LIN {X 0,Y 564.542,Z 419.185,A -85,B 0,C 180,E1 24922.898,E2 24922.898} C_VEL
LIN {X 0,Y 566.553,Z 422.727,A -85,B 0,C 180,E1 24922.507,E2 24922.507} C_VEL
LIN {X 0,Y 580.883,Z 441.824,A -85,B 0,C 180,E1 24920.03,E2 24920.03} C_VEL
LIN {X 0,Y 586.064,Z 449.548,A -85,B 0,C 180,E1 24919.171,E2 24919.171} C_VEL
LIN {X 0,Y 576.668,Z 659.273,A -85,B 0,C 180,E1 24915.972,E2 24915.972} C_VEL
LIN {X 0,Y 572.189,Z 766.018,A -85,B 0,C 180,E1 24914.357,E2 24914.357} C_VEL
LIN {X 0,Y 570.088,Z 794.768,A -85,B 0,C 180,E1 24913.761,E2 24913.761} C_VEL
LIN {X 0,Y 567.768,Z 818.372,A -85,B 0,C 180,E1 24913.108,E2 24913.108} C_VEL
LIN {X 0,Y 565.366,Z 838.963,A -85,B 0,C 180,E1 24912.414,E2 24912.414} C_VEL
LIN {X 0,Y 562.569,Z 859.83,A -85,B 0,C 180,E1 24911.584,E2 24911.584} C_VEL
LIN {X 0,Y 558.94,Z 883.872,A -85,B 0,C 180,E1 24910.457,E2 24910.457} C_VEL
LIN {X 0,Y 554.622,Z 908.25,A -85,B 0,C 180,E1 24909.087,E2 24909.087} C_VEL
LIN {X 0,Y 551.08,Z 926.843,A -85,B 0,C 180,E1 24907.884,E2 24907.884} C_VEL
LIN {X 0,Y 547.473,Z 944.537,A -85,B 0,C 180,E1 24906.595,E2 24906.595} C_VEL
LIN {X 0,Y 543.684,Z 962.173,A -85,B 0,C 180,E1 24905.151,E2 24905.151} C_VEL
LIN {X 0,Y 538.855,Z 983.671,A -85,B 0,C 180,E1 24903.145,E2 24903.145} C_VEL
LIN {X 0,Y 534.335,Z 1002.75,A -85,B 0,C 180,E1 24901.078,E2 24901.078} C_VEL
LIN {X 0,Y 530.36,Z 1019.387,A -85,B 0,C 180,E1 24899.024,E2 24899.024} C_VEL
LIN {X 0,Y 526.19,Z 1036.957,A -85,B 0,C 180,E1 24896.534,E2 24896.534} C_VEL
LIN {X 0,Y 522.376,Z 1053.129,A -85,B 0,C 180,E1 24893.876,E2 24893.876} C_VEL
LIN {X 0,Y 519.153,Z 1069.381,A -85,B 0,C 180,E1 24890.912,E2 24890.912} C_VEL
LIN {X 0,Y 516.803,Z 1082.675,A -85,B 0,C 180,E1 24888.127,E2 24888.127} C_VEL
LIN {X 0,Y 514.982,Z 1094.284,A -85,B 0,C 180,E1 24885.286,E2 24885.286} C_VEL
LIN {X 0,Y 513.617,Z 1104.724,A -85,B 0,C 180,E1 24882.289,E2 24882.289} C_VEL
LIN {X 0,Y 512.807,Z 1113.008,A -85,B 0,C 180,E1 24879.455,E2 24879.455} C_VEL
LIN {X 0,Y 512.269,Z 1120.002,A -85,B 0,C 180,E1 24876.47,E2 24876.47} C_VEL
LIN {X 0,Y 512.013,Z 1125.314,A -85,B 0,C 180,E1 24873.55,E2 24873.55} C_VEL
LIN {X 0,Y 511.941,Z 1128.909,A -85,B 0,C 180,E1 24870.779,E2 24870.779} C_VEL
LIN {X 0,Y 511.913,Z 1131.135,A -85,B 0,C 180,E1 24867.955,E2 24867.955} C_VEL
LIN {X 0,Y 511.904,Z 1131.984,A -85,B 0,C 180,E1 24865.079,E2 24865.079} C_VEL
LIN {X 0,Y 511.904,Z 1131.233,A -85,B 0,C 180,E1 24862.147,E2 24862.147} C_VEL
LIN {X 0,Y 511.939,Z 1129.064,A -85,B 0,C 180,E1 24859.274,E2 24859.274} C_VEL
LIN {X 0,Y 512.001,Z 1125.626,A -85,B 0,C 180,E1 24856.566,E2 24856.566} C_VEL
LIN {X 0,Y 512.205,Z 1120.709,A -85,B 0,C 180,E1 24853.778,E2 24853.778} C_VEL
LIN {X 0,Y 512.707,Z 1114.184,A -85,B 0,C 180,E1 24850.904,E2 24850.904} C_VEL
LIN {X 0,Y 513.531,Z 1105.747,A -85,B 0,C 180,E1 24847.946,E2 24847.946} C_VEL
LIN {X 0,Y 514.839,Z 1095.333,A -85,B 0,C 180,E1 24844.902,E2 24844.902} C_VEL
LIN {X 0,Y 516.649,Z 1083.593,A -85,B 0,C 180,E1 24841.996,E2 24841.996} C_VEL
LIN {X 0,Y 518.987,Z 1070.357,A -85,B 0,C 180,E1 24839.185,E2 24839.185} C_VEL
LIN {X 0,Y 523.302,Z 1049.733,A -85,B 0,C 180,E1 24835.397,E2 24835.397} C_VEL
LIN {X 0,Y 527.1,Z 1034.636,A -85,B 0,C 180,E1 24832.917,E2 24832.917} C_VEL
LIN {X 0,Y 530.836,Z 1019.658,A -85,B 0,C 180,E1 24830.787,E2 24830.787} C_VEL
LIN {X 0,Y 534.371,Z 1005.434,A -85,B 0,C 180,E1 24828.997,E2 24828.997} C_VEL
LIN {X 0,Y 537.967,Z 990.583,A -85,B 0,C 180,E1 24827.331,E2 24827.331} C_VEL
LIN {X 0,Y 542.61,Z 970.761,A -85,B 0,C 180,E1 24825.377,E2 24825.377} C_VEL
LIN {X 0,Y 546.709,Z 951.555,A -85,B 0,C 180,E1 24823.75,E2 24823.75} C_VEL
LIN {X 0,Y 550.21,Z 934.054,A -85,B 0,C 180,E1 24822.442,E2 24822.442} C_VEL
LIN {X 0,Y 553.849,Z 914.316,A -85,B 0,C 180,E1 24821.146,E2 24821.146} C_VEL
LIN {X 0,Y 557.856,Z 889.499,A -85,B 0,C 180,E1 24819.761,E2 24819.761} C_VEL
LIN {X 0,Y 560.615,Z 869.773,A -85,B 0,C 180,E1 24818.828,E2 24818.828} C_VEL
LIN {X 0,Y 562.93,Z 850.518,A -85,B 0,C 180,E1 24818.044,E2 24818.044} C_VEL
LIN {X 0,Y 565.079,Z 829.301,A -85,B 0,C 180,E1 24817.31,E2 24817.31} C_VEL
LIN {X 0,Y 567.288,Z 800.913,A -85,B 0,C 180,E1 24816.536,E2 24816.536} C_VEL
LIN {X 0,Y 568.472,Z 778.885,A -85,B 0,C 180,E1 24816.082,E2 24816.082} C_VEL
LIN {X 0,Y 574.153,Z 658.763,A -85,B 0,C 180,E1 24814.166,E2 24814.166} C_VEL
LIN {X 0,Y 579.443,Z 579.746,A -85,B 0,C 180,E1 24812.805,E2 24812.805} C_VEL
LIN {X 0,Y 586.189,Z 505.599,A -85,B 0,C 180,E1 24811.443,E2 24811.443} C_VEL
LIN {X 0,Y 592.771,Z 449.982,A -85,B 0,C 180,E1 24810.35,E2 24810.35} C_VEL
LIN {X 0,Y 591.734,Z 444.986,A -85,B 0,C 180,E1 24809.456,E2 24809.456} C_VEL
LIN {X 0,Y 591.658,Z 444.729,A -85,B 0,C 180,E1 24809.362,E2 24809.362} C_VEL
LIN {X 0,Y 589.852,Z 450.751,A -85,B 0,C 180,E1 24808.449,E2 24808.449} C_VEL
LIN {X 0,Y 588.941,Z 461.125,A -85,B 0,C 180,E1 24807.237,E2 24807.237} C_VEL
LIN {X 0,Y 589.012,Z 464.19,A -85,B 0,C 180,E1 24806.908,E2 24806.908} C_VEL
LIN {X 0,Y 588.095,Z 484.724,A -85,B 0,C 180,E1 24805.902,E2 24805.902} C_VEL
LIN {X 0,Y 588.06,Z 490.969,A -85,B 0,C 180,E1 24805.601,E2 24805.601} C_VEL
LIN {X 0,Y 581.292,Z 561.279,A -85,B 0,C 180,E1 24804.259,E2 24804.259} C_VEL
LIN {X 0,Y 575.759,Z 638.702,A -85,B 0,C 180,E1 24802.87,E2 24802.87} C_VEL
LIN {X 0,Y 570.578,Z 738.854,A -85,B 0,C 180,E1 24801.211,E2 24801.211} C_VEL
LIN {X 0,Y 565.248,Z 887.623,A -85,B 0,C 180,E1 24798.952,E2 24798.952} C_VEL
LIN {X 0,Y 563.149,Z 916.285,A -85,B 0,C 180,E1 24798.378,E2 24798.378} C_VEL
LIN {X 0,Y 560.931,Z 940.423,A -85,B 0,C 180,E1 24797.778,E2 24797.778} C_VEL
LIN {X 0,Y 558.001,Z 968.794,A -85,B 0,C 180,E1 24796.91,E2 24796.91} C_VEL
LIN {X 0,Y 554.811,Z 996.1,A -85,B 0,C 180,E1 24795.867,E2 24795.867} C_VEL
LIN {X 0,Y 552.139,Z 1017.393,A -85,B 0,C 180,E1 24794.921,E2 24794.921} C_VEL
LIN {X 0,Y 549.242,Z 1038.814,A -85,B 0,C 180,E1 24793.843,E2 24793.843} C_VEL
LIN {X 0,Y 546.178,Z 1060.331,A -85,B 0,C 180,E1 24792.613,E2 24792.613} C_VEL
LIN {X 0,Y 542.506,Z 1085.129,A -85,B 0,C 180,E1 24791.005,E2 24791.005} C_VEL
LIN {X 0,Y 538.667,Z 1108.867,A -85,B 0,C 180,E1 24789.22,E2 24789.22} C_VEL
LIN {X 0,Y 535.764,Z 1126.329,A -85,B 0,C 180,E1 24787.744,E2 24787.744} C_VEL
LIN {X 0,Y 533.088,Z 1142.045,A -85,B 0,C 180,E1 24786.282,E2 24786.282} C_VEL
LIN {X 0,Y 530.41,Z 1157.572,A -85,B 0,C 180,E1 24784.701,E2 24784.701} C_VEL
LIN {X 0,Y 527.7,Z 1173.227,A -85,B 0,C 180,E1 24782.943,E2 24782.943} C_VEL
LIN {X 0,Y 525.229,Z 1187.423,A -85,B 0,C 180,E1 24781.185,E2 24781.185} C_VEL
LIN {X 0,Y 523.309,Z 1198.436,A -85,B 0,C 180,E1 24779.661,E2 24779.661} C_VEL
LIN {X 0,Y 520.705,Z 1211.245,A -85,B 0,C 180,E1 24777.481,E2 24777.481} C_VEL
LIN {X 0,Y 518.448,Z 1222.98,A -85,B 0,C 180,E1 24775.228,E2 24775.228} C_VEL
LIN {X 0,Y 516.666,Z 1233.28,A -85,B 0,C 180,E1 24773.012,E2 24773.012} C_VEL
LIN {X 0,Y 515.063,Z 1243.808,A -85,B 0,C 180,E1 24770.452,E2 24770.452} C_VEL
LIN {X 0,Y 513.624,Z 1254.739,A -85,B 0,C 180,E1 24767.328,E2 24767.328} C_VEL
LIN {X 0,Y 512.851,Z 1262.137,A -85,B 0,C 180,E1 24764.797,E2 24764.797} C_VEL
LIN {X 0,Y 512.406,Z 1267.799,A -85,B 0,C 180,E1 24762.509,E2 24762.509} C_VEL
LIN {X 0,Y 512.121,Z 1272.693,A -85,B 0,C 180,E1 24760.12,E2 24760.12} C_VEL
LIN {X 0,Y 511.965,Z 1276.677,A -85,B 0,C 180,E1 24757.632,E2 24757.632} C_VEL
LIN {X 0,Y 511.924,Z 1279.659,A -85,B 0,C 180,E1 24755.038,E2 24755.038} C_VEL
LIN {X 0,Y 511.911,Z 1281.599,A -85,B 0,C 180,E1 24752.015,E2 24752.015} C_VEL
LIN {X 0,Y 511.865,Z 1281.871,A -85,B 0,C 180,E1 24749.328,E2 24749.328} C_VEL
LIN {X 0,Y 511.909,Z 1281.082,A -85,B 0,C 180,E1 24746.977,E2 24746.977} C_VEL
LIN {X 0,Y 511.93,Z 1279.199,A -85,B 0,C 180,E1 24744.508,E2 24744.508} C_VEL
LIN {X 0,Y 511.97,Z 1276.356,A -85,B 0,C 180,E1 24742.142,E2 24742.142} C_VEL
LIN {X 0,Y 512.156,Z 1272.279,A -85,B 0,C 180,E1 24739.653,E2 24739.653} C_VEL
LIN {X 0,Y 512.544,Z 1266.27,A -85,B 0,C 180,E1 24736.806,E2 24736.806} C_VEL
LIN {X 0,Y 513.279,Z 1257.914,A -85,B 0,C 180,E1 24733.709,E2 24733.709} C_VEL
LIN {X 0,Y 514.226,Z 1249.696,A -85,B 0,C 180,E1 24731.169,E2 24731.169} C_VEL
LIN {X 0,Y 515.454,Z 1241.06,A -85,B 0,C 180,E1 24728.851,E2 24728.851} C_VEL
LIN {X 0,Y 517.115,Z 1230.712,A -85,B 0,C 180,E1 24726.406,E2 24726.406} C_VEL
LIN {X 0,Y 519.818,Z 1215.891,A -85,B 0,C 180,E1 24723.373,E2 24723.373} C_VEL
LIN {X 0,Y 522.446,Z 1202.553,A -85,B 0,C 180,E1 24721.002,E2 24721.002} C_VEL
LIN {X 0,Y 524.453,Z 1192.013,A -85,B 0,C 180,E1 24719.4,E2 24719.4} C_VEL
LIN {X 0,Y 527.516,Z 1175.905,A -85,B 0,C 180,E1 24717.238,E2 24717.238} C_VEL
LIN {X 0,Y 530.602,Z 1160.006,A -85,B 0,C 180,E1 24715.313,E2 24715.313} C_VEL
LIN {X 0,Y 534.437,Z 1140.647,A -85,B 0,C 180,E1 24713.203,E2 24713.203} C_VEL
LIN {X 0,Y 538.764,Z 1118.423,A -85,B 0,C 180,E1 24711.082,E2 24711.082} C_VEL
LIN {X 0,Y 542.437,Z 1099.473,A -85,B 0,C 180,E1 24709.476,E2 24709.476} C_VEL
LIN {X 0,Y 546.072,Z 1080.345,A -85,B 0,C 180,E1 24708.023,E2 24708.023} C_VEL
LIN {X 0,Y 550.322,Z 1057.451,A -85,B 0,C 180,E1 24706.48,E2 24706.48} C_VEL
LIN {X 0,Y 554.631,Z 1032.424,A -85,B 0,C 180,E1 24705.034,E2 24705.034} C_VEL
LIN {X 0,Y 558.14,Z 1010.377,A -85,B 0,C 180,E1 24703.932,E2 24703.932} C_VEL
LIN {X 0,Y 561.113,Z 990.283,A -85,B 0,C 180,E1 24703.063,E2 24703.063} C_VEL
LIN {X 0,Y 564.037,Z 968.586,A -85,B 0,C 180,E1 24702.259,E2 24702.259} C_VEL
LIN {X 0,Y 567.292,Z 941.486,A -85,B 0,C 180,E1 24701.432,E2 24701.432} C_VEL
LIN {X 0,Y 569.778,Z 915.224,A -85,B 0,C 180,E1 24700.824,E2 24700.824} C_VEL
LIN {X 0,Y 571.357,Z 892.816,A -85,B 0,C 180,E1 24700.418,E2 24700.418} C_VEL
LIN {X 0,Y 580.407,Z 670.692,A -85,B 0,C 180,E1 24697.065,E2 24697.065} C_VEL
LIN {X 0,Y 588.793,Z 490.152,A -85,B 0,C 180,E1 24694.268,E2 24694.268} C_VEL
LIN {X 0,Y 585.464,Z 469.461,A -85,B 0,C 180,E1 24693.362,E2 24693.362} C_VEL
LIN {X 0,Y 573.553,Z 450.96,A -85,B 0,C 180,E1 24691.241,E2 24691.241} C_VEL
LIN {X 0,Y 560.617,Z 432.091,A -85,B 0,C 180,E1 24688.758,E2 24688.758} C_VEL
LIN {X 0,Y 549.882,Z 417.05,A -85,B 0,C 180,E1 24686.514,E2 24686.514} C_VEL
LIN {X 0,Y 542.341,Z 406.72,A -85,B 0,C 180,E1 24684.828,E2 24684.828} C_VEL
LIN {X 0,Y 539.641,Z 402.462,A -85,B 0,C 180,E1 24684.056,E2 24684.056} C_VEL
LIN {X 0,Y 534.084,Z 392.609,A -85,B 0,C 180,E1 24681.874,E2 24681.874} C_VEL
LIN {X 0,Y 531.056,Z 387.284,A -85,B 0,C 180,E1 24680.615,E2 24680.615} C_VEL
LIN {X 0,Y 528.6,Z 382.928,A -85,B 0,C 180,E1 24679.561,E2 24679.561} C_VEL
LIN {X 0,Y 525.714,Z 377.911,A -85,B 0,C 180,E1 24678.29,E2 24678.29} C_VEL
LIN {X 0,Y 523.432,Z 373.779,A -85,B 0,C 180,E1 24677.223,E2 24677.223} C_VEL
LIN {X 0,Y 520.587,Z 369.323,A -85,B 0,C 180,E1 24675.942,E2 24675.942} C_VEL
LIN {X 0,Y 519.744,Z 367.693,A -85,B 0,C 180,E1 24675.51,E2 24675.51} C_VEL
LIN {X 0,Y 517.472,Z 364.139,A -85,B 0,C 180,E1 24674.434,E2 24674.434} C_VEL
LIN {X 0,Y 516.444,Z 362.289,A -85,B 0,C 180,E1 24673.891,E2 24673.891} C_VEL
LIN {X 0,Y 514.205,Z 358.902,A -85,B 0,C 180,E1 24672.808,E2 24672.808} C_VEL
LIN {X 0,Y 513.815,Z 357.412,A -85,B 0,C 180,E1 24672.344,E2 24672.344} C_VEL
LIN {X 0,Y 513.806,Z 357.208,A -85,B 0,C 180,E1 24668.956,E2 24668.956} C_VEL
LIN {X 0,Y 513.781,Z 357.211,A -85,B 0,C 180,E1 24665.584,E2 24665.584} C_VEL
LIN {X 0,Y 513.782,Z 357.21,A -85,B 0,C 180,E1 24662.007,E2 24662.007} C_VEL
LIN {X 0,Y 513.81,Z 357.225,A -85,B 0,C 180,E1 24658.662,E2 24658.662} C_VEL
LIN {X 0,Y 513.782,Z 357.226,A -85,B 0,C 180,E1 24655.2,E2 24655.2} C_VEL
LIN {X 0,Y 513.781,Z 357.229,A -85,B 0,C 180,E1 24651.72,E2 24651.72} C_VEL
LIN {X 0,Y 513.81,Z 357.23,A -85,B 0,C 180,E1 24648.323,E2 24648.323} C_VEL
LIN {X 0,Y 513.776,Z 357.23,A -85,B 0,C 180,E1 24644.883,E2 24644.883} C_VEL
LIN {X 0,Y 513.778,Z 357.235,A -85,B 0,C 180,E1 24641.387,E2 24641.387} C_VEL
LIN {X 0,Y 513.815,Z 357.229,A -85,B 0,C 180,E1 24637.94,E2 24637.94} C_VEL
LIN {X 0,Y 513.777,Z 357.231,A -85,B 0,C 180,E1 24634.526,E2 24634.526} C_VEL
LIN {X 0,Y 513.769,Z 357.223,A -85,B 0,C 180,E1 24631.013,E2 24631.013} C_VEL
LIN {X 0,Y 513.81,Z 357.218,A -85,B 0,C 180,E1 24627.625,E2 24627.625} C_VEL
LIN {X 0,Y 513.767,Z 357.22,A -85,B 0,C 180,E1 24624.248,E2 24624.248} C_VEL
LIN {X 0,Y 513.766,Z 357.223,A -85,B 0,C 180,E1 24620.764,E2 24620.764} C_VEL
LIN {X 0,Y 513.805,Z 357.216,A -85,B 0,C 180,E1 24617.522,E2 24617.522} C_VEL
LIN {X 0,Y 513.757,Z 357.227,A -85,B 0,C 180,E1 24614.097,E2 24614.097} C_VEL
LIN {X 0,Y 513.771,Z 357.229,A -85,B 0,C 180,E1 24610.623,E2 24610.623} C_VEL
LIN {X 0,Y 513.785,Z 357.228,A -85,B 0,C 180,E1 24607.386,E2 24607.386} C_VEL
LIN {X 0,Y 513.749,Z 357.236,A -85,B 0,C 180,E1 24603.957,E2 24603.957} C_VEL
LIN {X 0,Y 513.786,Z 357.228,A -85,B 0,C 180,E1 24600.526,E2 24600.526} C_VEL
LIN {X 0,Y 513.759,Z 357.229,A -85,B 0,C 180,E1 24597.342,E2 24597.342} C_VEL
LIN {X 0,Y 513.745,Z 357.22,A -85,B 0,C 180,E1 24593.829,E2 24593.829} C_VEL
LIN {X 0,Y 513.804,Z 357.216,A -85,B 0,C 180,E1 24590.505,E2 24590.505} C_VEL
LIN {X 0,Y 513.746,Z 357.229,A -85,B 0,C 180,E1 24587.133,E2 24587.133} C_VEL
LIN {X 0,Y 513.745,Z 357.238,A -85,B 0,C 180,E1 24583.621,E2 24583.621} C_VEL
LIN {X 0,Y 513.791,Z 357.222,A -85,B 0,C 180,E1 24580.314,E2 24580.314} C_VEL
LIN {X 0,Y 513.729,Z 357.229,A -85,B 0,C 180,E1 24577.043,E2 24577.043} C_VEL
LIN {X 0,Y 513.77,Z 357.426,A -85,B 0,C 180,E1 24574.633,E2 24574.633} C_VEL
LIN {X 0,Y 514.096,Z 358.692,A -85,B 0,C 180,E1 24574.294,E2 24574.294} C_VEL
LIN {X 0,Y 516.027,Z 361.881,A -85,B 0,C 180,E1 24573.708,E2 24573.708} C_VEL
LIN {X 0,Y 519.046,Z 364.127,A -85,B 0,C 180,E1 24572.926,E2 24572.926} C_VEL
LIN {X 0,Y 521.208,Z 367.728,A -85,B 0,C 180,E1 24572.309,E2 24572.309} C_VEL
LIN {X 0,Y 524.346,Z 370.575,A -85,B 0,C 180,E1 24571.53,E2 24571.53} C_VEL
LIN {X 0,Y 527.134,Z 374.495,A -85,B 0,C 180,E1 24570.815,E2 24570.815} C_VEL
LIN {X 0,Y 529.519,Z 376.785,A -85,B 0,C 180,E1 24570.243,E2 24570.243} C_VEL
LIN {X 0,Y 532.724,Z 381.001,A -85,B 0,C 180,E1 24569.462,E2 24569.462} C_VEL
LIN {X 0,Y 534.849,Z 383.089,A -85,B 0,C 180,E1 24568.982,E2 24568.982} C_VEL
LIN {X 0,Y 538.583,Z 387.619,A -85,B 0,C 180,E1 24568.138,E2 24568.138} C_VEL
LIN {X 0,Y 544.66,Z 395.284,A -85,B 0,C 180,E1 24566.79,E2 24566.79} C_VEL
LIN {X 0,Y 550.439,Z 402.324,A -85,B 0,C 180,E1 24565.592,E2 24565.592} C_VEL
LIN {X 0,Y 558.593,Z 412.587,A -85,B 0,C 180,E1 24563.989,E2 24563.989} C_VEL
LIN {X 0,Y 566.553,Z 422.727,A -85,B 0,C 180,E1 24562.507,E2 24562.507} C_VEL
LIN {X 0,Y 569.307,Z 427.772,A -85,B 0,C 180,E1 24561.981,E2 24561.981} C_VEL
LIN {X 0,Y 575.605,Z 444.913,A -85,B 0,C 180,E1 24560.687,E2 24560.687} C_VEL
LIN {X 0,Y 577.65,Z 448.551,A -85,B 0,C 180,E1 24560.32,E2 24560.32} C_VEL
LIN {X 0,Y 581.063,Z 453.836,A -85,B 0,C 180,E1 24559.738,E2 24559.738} C_VEL
LIN {X 0,Y 571.594,Z 655.779,A -85,B 0,C 180,E1 24556.634,E2 24556.634} C_VEL
LIN {X 0,Y 566.718,Z 766.809,A -85,B 0,C 180,E1 24554.939,E2 24554.939} C_VEL
LIN {X 0,Y 564.563,Z 795.501,A -85,B 0,C 180,E1 24554.34,E2 24554.34} C_VEL
LIN {X 0,Y 562.139,Z 819.411,A -85,B 0,C 180,E1 24553.674,E2 24553.674} C_VEL
LIN {X 0,Y 559.605,Z 840.412,A -85,B 0,C 180,E1 24552.961,E2 24552.961} C_VEL
LIN {X 0,Y 556.484,Z 862.887,A -85,B 0,C 180,E1 24552.052,E2 24552.052} C_VEL
LIN {X 0,Y 552.17,Z 889.566,A -85,B 0,C 180,E1 24550.758,E2 24550.758} C_VEL
LIN {X 0,Y 548.427,Z 910.156,A -85,B 0,C 180,E1 24549.575,E2 24549.575} C_VEL
LIN {X 0,Y 544.737,Z 928.843,A -85,B 0,C 180,E1 24548.35,E2 24548.35} C_VEL
LIN {X 0,Y 541.011,Z 946.471,A -85,B 0,C 180,E1 24547.048,E2 24547.048} C_VEL
LIN {X 0,Y 536.434,Z 967.136,A -85,B 0,C 180,E1 24545.322,E2 24545.322} C_VEL
LIN {X 0,Y 531.518,Z 987.698,A -85,B 0,C 180,E1 24543.326,E2 24543.326} C_VEL
LIN {X 0,Y 527.397,Z 1004.566,A -85,B 0,C 180,E1 24541.461,E2 24541.461} C_VEL
LIN {X 0,Y 523.169,Z 1021.68,A -85,B 0,C 180,E1 24539.317,E2 24539.317} C_VEL
LIN {X 0,Y 518.813,Z 1039.305,A -85,B 0,C 180,E1 24536.766,E2 24536.766} C_VEL
LIN {X 0,Y 515.015,Z 1054.732,A -85,B 0,C 180,E1 24534.179,E2 24534.179} C_VEL
LIN {X 0,Y 511.728,Z 1068.988,A -85,B 0,C 180,E1 24531.406,E2 24531.406} C_VEL
LIN {X 0,Y 509.094,Z 1082.911,A -85,B 0,C 180,E1 24528.444,E2 24528.444} C_VEL
LIN {X 0,Y 507.153,Z 1094.564,A -85,B 0,C 180,E1 24525.538,E2 24525.538} C_VEL
LIN {X 0,Y 505.732,Z 1104.793,A -85,B 0,C 180,E1 24522.546,E2 24522.546} C_VEL
LIN {X 0,Y 504.859,Z 1113.219,A -85,B 0,C 180,E1 24519.609,E2 24519.609} C_VEL
LIN {X 0,Y 504.294,Z 1120.152,A -85,B 0,C 180,E1 24516.582,E2 24516.582} C_VEL
LIN {X 0,Y 504.017,Z 1125.479,A -85,B 0,C 180,E1 24513.571,E2 24513.571} C_VEL
LIN {X 0,Y 503.941,Z 1129.007,A -85,B 0,C 180,E1 24510.782,E2 24510.782} C_VEL
LIN {X 0,Y 503.911,Z 1131.172,A -85,B 0,C 180,E1 24507.923,E2 24507.923} C_VEL
LIN {X 0,Y 503.901,Z 1131.999,A -85,B 0,C 180,E1 24504.932,E2 24504.932} C_VEL
LIN {X 0,Y 503.915,Z 1131.196,A -85,B 0,C 180,E1 24502.026,E2 24502.026} C_VEL
LIN {X 0,Y 503.939,Z 1128.982,A -85,B 0,C 180,E1 24499.11,E2 24499.11} C_VEL
LIN {X 0,Y 504.023,Z 1125.524,A -85,B 0,C 180,E1 24496.362,E2 24496.362} C_VEL
LIN {X 0,Y 504.267,Z 1120.327,A -85,B 0,C 180,E1 24493.415,E2 24493.415} C_VEL
LIN {X 0,Y 504.844,Z 1113.426,A -85,B 0,C 180,E1 24490.383,E2 24490.383} C_VEL
LIN {X 0,Y 505.745,Z 1104.873,A -85,B 0,C 180,E1 24487.384,E2 24487.384} C_VEL
LIN {X 0,Y 507.132,Z 1094.7,A -85,B 0,C 180,E1 24484.41,E2 24484.41} C_VEL
LIN {X 0,Y 509.098,Z 1082.793,A -85,B 0,C 180,E1 24481.449,E2 24481.449} C_VEL
LIN {X 0,Y 512.682,Z 1065.064,A -85,B 0,C 180,E1 24477.653,E2 24477.653} C_VEL
LIN {X 0,Y 516.376,Z 1050.682,A -85,B 0,C 180,E1 24474.89,E2 24474.89} C_VEL
LIN {X 0,Y 520.531,Z 1034.687,A -85,B 0,C 180,E1 24472.272,E2 24472.272} C_VEL
LIN {X 0,Y 524.058,Z 1021.117,A -85,B 0,C 180,E1 24470.334,E2 24470.334} C_VEL
LIN {X 0,Y 527.729,Z 1006.863,A -85,B 0,C 180,E1 24468.525,E2 24468.525} C_VEL
LIN {X 0,Y 531.96,Z 990.047,A -85,B 0,C 180,E1 24466.633,E2 24466.633} C_VEL
LIN {X 0,Y 536.78,Z 969.736,A -85,B 0,C 180,E1 24464.662,E2 24464.662} C_VEL
LIN {X 0,Y 540.507,Z 952.834,A -85,B 0,C 180,E1 24463.227,E2 24463.227} C_VEL
LIN {X 0,Y 544.126,Z 935.295,A -85,B 0,C 180,E1 24461.907,E2 24461.907} C_VEL
LIN {X 0,Y 548.189,Z 913.913,A -85,B 0,C 180,E1 24460.501,E2 24460.501} C_VEL
LIN {X 0,Y 552.006,Z 890.549,A -85,B 0,C 180,E1 24459.205,E2 24459.205} C_VEL
LIN {X 0,Y 554.846,Z 870.735,A -85,B 0,C 180,E1 24458.264,E2 24458.264} C_VEL
LIN {X 0,Y 557.385,Z 850.097,A -85,B 0,C 180,E1 24457.425,E2 24457.425} C_VEL
LIN {X 0,Y 560.062,Z 823.338,A -85,B 0,C 180,E1 24456.532,E2 24456.532} C_VEL
LIN {X 0,Y 561.793,Z 799.943,A -85,B 0,C 180,E1 24455.922,E2 24455.922} C_VEL
LIN {X 0,Y 562.966,Z 778.302,A -85,B 0,C 180,E1 24455.481,E2 24455.481} C_VEL
LIN {X 0,Y 568.565,Z 670.891,A -85,B 0,C 180,E1 24453.728,E2 24453.728} C_VEL
LIN {X 0,Y 574.051,Z 595.784,A -85,B 0,C 180,E1 24452.405,E2 24452.405} C_VEL
LIN {X 0,Y 581.095,Z 524.407,A -85,B 0,C 180,E1 24451.067,E2 24451.067} C_VEL
LIN {X 0,Y 589.015,Z 463.58,A -85,B 0,C 180,E1 24449.874,E2 24449.874} C_VEL
LIN {X 0,Y 590.299,Z 454.826,A -85,B 0,C 180,E1 24449.684,E2 24449.684} C_VEL
LIN {X 0,Y 590.055,Z 453.628,A -85,B 0,C 180,E1 24449.41,E2 24449.41} C_VEL
LIN {X 0,Y 588.383,Z 458.932,A -85,B 0,C 180,E1 24448.698,E2 24448.698} C_VEL
LIN {X 0,Y 587.017,Z 469.009,A -85,B 0,C 180,E1 24447.521,E2 24447.521} C_VEL
LIN {X 0,Y 585.338,Z 488.257,A -85,B 0,C 180,E1 24446.549,E2 24446.549} C_VEL
LIN {X 0,Y 585.073,Z 493.464,A -85,B 0,C 180,E1 24446.296,E2 24446.296} C_VEL
LIN {X 0,Y 577.832,Z 557.664,A -85,B 0,C 180,E1 24445.031,E2 24445.031} C_VEL
LIN {X 0,Y 571.755,Z 628.875,A -85,B 0,C 180,E1 24443.699,E2 24443.699} C_VEL
LIN {X 0,Y 566.38,Z 714.472,A -85,B 0,C 180,E1 24442.21,E2 24442.21} C_VEL
LIN {X 0,Y 561.972,Z 814.359,A -85,B 0,C 180,E1 24440.62,E2 24440.62} C_VEL
LIN {X 0,Y 559.245,Z 885.059,A -85,B 0,C 180,E1 24439.522,E2 24439.522} C_VEL
LIN {X 0,Y 557.025,Z 913.922,A -85,B 0,C 180,E1 24438.936,E2 24438.936} C_VEL
LIN {X 0,Y 554.653,Z 938.566,A -85,B 0,C 180,E1 24438.318,E2 24438.318} C_VEL
LIN {X 0,Y 551.445,Z 967.947,A -85,B 0,C 180,E1 24437.405,E2 24437.405} C_VEL
LIN {X 0,Y 548.243,Z 994.278,A -85,B 0,C 180,E1 24436.389,E2 24436.389} C_VEL
LIN {X 0,Y 545.394,Z 1016.007,A -85,B 0,C 180,E1 24435.417,E2 24435.417} C_VEL
LIN {X 0,Y 542.227,Z 1038.62,A -85,B 0,C 180,E1 24434.263,E2 24434.263} C_VEL
LIN {X 0,Y 538.414,Z 1064.669,A -85,B 0,C 180,E1 24432.738,E2 24432.738} C_VEL
LIN {X 0,Y 534.511,Z 1089.022,A -85,B 0,C 180,E1 24431.072,E2 24431.072} C_VEL
LIN {X 0,Y 531.398,Z 1107.76,A -85,B 0,C 180,E1 24429.632,E2 24429.632} C_VEL
LIN {X 0,Y 528.323,Z 1125.809,A -85,B 0,C 180,E1 24428.095,E2 24428.095} C_VEL
LIN {X 0,Y 525.387,Z 1142.545,A -85,B 0,C 180,E1 24426.51,E2 24426.51} C_VEL
LIN {X 0,Y 522.713,Z 1157.472,A -85,B 0,C 180,E1 24424.953,E2 24424.953} C_VEL
LIN {X 0,Y 520.342,Z 1170.835,A -85,B 0,C 180,E1 24423.433,E2 24423.433} C_VEL
LIN {X 0,Y 517.822,Z 1184.912,A -85,B 0,C 180,E1 24421.682,E2 24421.682} C_VEL
LIN {X 0,Y 515.384,Z 1198.765,A -85,B 0,C 180,E1 24419.779,E2 24419.779} C_VEL
LIN {X 0,Y 513.335,Z 1210.474,A -85,B 0,C 180,E1 24417.997,E2 24417.997} C_VEL
LIN {X 0,Y 511.442,Z 1220.274,A -85,B 0,C 180,E1 24416.186,E2 24416.186} C_VEL
LIN {X 0,Y 509.278,Z 1231.735,A -85,B 0,C 180,E1 24413.733,E2 24413.733} C_VEL
LIN {X 0,Y 507.58,Z 1241.838,A -85,B 0,C 180,E1 24411.287,E2 24411.287} C_VEL
LIN {X 0,Y 506.243,Z 1250.911,A -85,B 0,C 180,E1 24408.78,E2 24408.78} C_VEL
LIN {X 0,Y 505.116,Z 1260.622,A -85,B 0,C 180,E1 24405.617,E2 24405.617} C_VEL
LIN {X 0,Y 504.466,Z 1267.622,A -85,B 0,C 180,E1 24402.79,E2 24402.79} C_VEL
LIN {X 0,Y 504.149,Z 1272.69,A -85,B 0,C 180,E1 24400.282,E2 24400.282} C_VEL
LIN {X 0,Y 503.969,Z 1276.674,A -85,B 0,C 180,E1 24397.753,E2 24397.753} C_VEL
LIN {X 0,Y 503.925,Z 1279.651,A -85,B 0,C 180,E1 24395.123,E2 24395.123} C_VEL
LIN {X 0,Y 503.911,Z 1281.599,A -85,B 0,C 180,E1 24392.047,E2 24392.047} C_VEL
LIN {X 0,Y 503.865,Z 1281.871,A -85,B 0,C 180,E1 24389.318,E2 24389.318} C_VEL
LIN {X 0,Y 503.909,Z 1281.081,A -85,B 0,C 180,E1 24386.929,E2 24386.929} C_VEL
LIN {X 0,Y 503.93,Z 1279.309,A -85,B 0,C 180,E1 24384.535,E2 24384.535} C_VEL
LIN {X 0,Y 503.972,Z 1276.513,A -85,B 0,C 180,E1 24382.132,E2 24382.132} C_VEL
LIN {X 0,Y 504.167,Z 1272.483,A -85,B 0,C 180,E1 24379.603,E2 24379.603} C_VEL
LIN {X 0,Y 504.496,Z 1267.289,A -85,B 0,C 180,E1 24377.058,E2 24377.058} C_VEL
LIN {X 0,Y 505.208,Z 1259.679,A -85,B 0,C 180,E1 24374.032,E2 24374.032} C_VEL
LIN {X 0,Y 506.298,Z 1250.437,A -85,B 0,C 180,E1 24371.082,E2 24371.082} C_VEL
LIN {X 0,Y 507.58,Z 1241.841,A -85,B 0,C 180,E1 24368.713,E2 24368.713} C_VEL
LIN {X 0,Y 509.28,Z 1231.74,A -85,B 0,C 180,E1 24366.267,E2 24366.267} C_VEL
LIN {X 0,Y 511.856,Z 1218.395,A -85,B 0,C 180,E1 24363.427,E2 24363.427} C_VEL
LIN {X 0,Y 514.237,Z 1205.468,A -85,B 0,C 180,E1 24361.17,E2 24361.17} C_VEL
LIN {X 0,Y 517.24,Z 1189.722,A -85,B 0,C 180,E1 24358.797,E2 24358.797} C_VEL
LIN {X 0,Y 520.189,Z 1174.881,A -85,B 0,C 180,E1 24356.783,E2 24356.783} C_VEL
LIN {X 0,Y 523.355,Z 1159.197,A -85,B 0,C 180,E1 24354.857,E2 24354.857} C_VEL
LIN {X 0,Y 527.237,Z 1140.364,A -85,B 0,C 180,E1 24352.774,E2 24352.774} C_VEL
LIN {X 0,Y 531.932,Z 1117.444,A -85,B 0,C 180,E1 24350.555,E2 24350.555} C_VEL
LIN {X 0,Y 535.761,Z 1098.517,A -85,B 0,C 180,E1 24348.934,E2 24348.934} C_VEL
LIN {X 0,Y 539.462,Z 1079.841,A -85,B 0,C 180,E1 24347.5,E2 24347.5} C_VEL
LIN {X 0,Y 543.629,Z 1058.257,A -85,B 0,C 180,E1 24346.027,E2 24346.027} C_VEL
LIN {X 0,Y 548.275,Z 1032.596,A -85,B 0,C 180,E1 24344.516,E2 24344.516} C_VEL
LIN {X 0,Y 551.898,Z 1010.611,A -85,B 0,C 180,E1 24343.407,E2 24343.407} C_VEL
LIN {X 0,Y 555.141,Z 989.524,A -85,B 0,C 180,E1 24342.488,E2 24342.488} C_VEL
LIN {X 0,Y 558.096,Z 968.434,A -85,B 0,C 180,E1 24341.7,E2 24341.7} C_VEL
LIN {X 0,Y 561.331,Z 942.78,A -85,B 0,C 180,E1 24340.904,E2 24340.904} C_VEL
LIN {X 0,Y 564.099,Z 915.16,A -85,B 0,C 180,E1 24340.25,E2 24340.25} C_VEL
LIN {X 0,Y 565.78,Z 892.4,A -85,B 0,C 180,E1 24339.832,E2 24339.832} C_VEL
LIN {X 0,Y 575.419,Z 666.099,A -85,B 0,C 180,E1 24336.388,E2 24336.388} C_VEL
LIN {X 0,Y 583.885,Z 492.052,A -85,B 0,C 180,E1 24333.666,E2 24333.666} C_VEL
LIN {X 0,Y 581.088,Z 474.396,A -85,B 0,C 180,E1 24332.881,E2 24332.881} C_VEL
LIN {X 0,Y 569.439,Z 456.296,A -85,B 0,C 180,E1 24330.758,E2 24330.758} C_VEL
LIN {X 0,Y 557.306,Z 438.453,A -85,B 0,C 180,E1 24328.389,E2 24328.389} C_VEL
LIN {X 0,Y 546.847,Z 423.716,A -85,B 0,C 180,E1 24326.175,E2 24326.175} C_VEL
LIN {X 0,Y 536.869,Z 409.782,A -85,B 0,C 180,E1 24323.867,E2 24323.867} C_VEL
LIN {X 0,Y 530.604,Z 401.174,A -85,B 0,C 180,E1 24322.258,E2 24322.258} C_VEL
LIN {X 0,Y 526.007,Z 393.127,A -85,B 0,C 180,E1 24320.357,E2 24320.357} C_VEL
LIN {X 0,Y 523.8,Z 389.169,A -85,B 0,C 180,E1 24319.399,E2 24319.399} C_VEL
LIN {X 0,Y 520.669,Z 383.816,A -85,B 0,C 180,E1 24318.01,E2 24318.01} C_VEL
LIN {X 0,Y 518.167,Z 379.32,A -85,B 0,C 180,E1 24316.825,E2 24316.825} C_VEL
LIN {X 0,Y 515.842,Z 375.52,A -85,B 0,C 180,E1 24315.746,E2 24315.746} C_VEL
LIN {X 0,Y 514.713,Z 373.662,A -85,B 0,C 180,E1 24315.204,E2 24315.204} C_VEL
LIN {X 0,Y 512.421,Z 369.442,A -85,B 0,C 180,E1 24314.002,E2 24314.002} C_VEL
LIN {X 0,Y 509.7,Z 365.51,A -85,B 0,C 180,E1 24312.692,E2 24312.692} C_VEL
LIN {X 0,Y 508.785,Z 363.536,A -85,B 0,C 180,E1 24312.139,E2 24312.139} C_VEL
LIN {X 0,Y 506.38,Z 360.193,A -85,B 0,C 180,E1 24310.927,E2 24310.927} C_VEL
LIN {X 0,Y 505.882,Z 358.418,A -85,B 0,C 180,E1 24310.362,E2 24310.362} C_VEL
LIN {X 0,Y 505.872,Z 358.218,A -85,B 0,C 180,E1 24307.039,E2 24307.039} C_VEL
LIN {X 0,Y 505.844,Z 358.223,A -85,B 0,C 180,E1 24303.513,E2 24303.513} C_VEL
LIN {X 0,Y 505.844,Z 358.224,A -85,B 0,C 180,E1 24299.887,E2 24299.887} C_VEL
LIN {X 0,Y 505.868,Z 358.217,A -85,B 0,C 180,E1 24296.374,E2 24296.374} C_VEL
LIN {X 0,Y 505.862,Z 358.214,A -85,B 0,C 180,E1 24292.847,E2 24292.847} C_VEL
LIN {X 0,Y 505.834,Z 358.217,A -85,B 0,C 180,E1 24289.407,E2 24289.407} C_VEL
LIN {X 0,Y 505.873,Z 358.216,A -85,B 0,C 180,E1 24285.929,E2 24285.929} C_VEL
LIN {X 0,Y 505.863,Z 358.205,A -85,B 0,C 180,E1 24282.397,E2 24282.397} C_VEL
LIN {X 0,Y 505.83,Z 358.216,A -85,B 0,C 180,E1 24278.908,E2 24278.908} C_VEL
LIN {X 0,Y 505.848,Z 358.219,A -85,B 0,C 180,E1 24275.402,E2 24275.402} C_VEL
LIN {X 0,Y 505.875,Z 358.218,A -85,B 0,C 180,E1 24271.938,E2 24271.938} C_VEL
LIN {X 0,Y 505.827,Z 358.222,A -85,B 0,C 180,E1 24268.543,E2 24268.543} C_VEL
LIN {X 0,Y 505.837,Z 358.214,A -85,B 0,C 180,E1 24265.023,E2 24265.023} C_VEL
LIN {X 0,Y 505.874,Z 358.207,A -85,B 0,C 180,E1 24261.509,E2 24261.509} C_VEL
LIN {X 0,Y 505.821,Z 358.211,A -85,B 0,C 180,E1 24258.179,E2 24258.179} C_VEL
LIN {X 0,Y 505.829,Z 358.21,A -85,B 0,C 180,E1 24254.632,E2 24254.632} C_VEL
LIN {X 0,Y 505.88,Z 358.204,A -85,B 0,C 180,E1 24251.143,E2 24251.143} C_VEL
LIN {X 0,Y 505.82,Z 358.216,A -85,B 0,C 180,E1 24247.748,E2 24247.748} C_VEL
LIN {X 0,Y 505.815,Z 358.226,A -85,B 0,C 180,E1 24244.153,E2 24244.153} C_VEL
LIN {X 0,Y 505.869,Z 358.217,A -85,B 0,C 180,E1 24240.704,E2 24240.704} C_VEL
LIN {X 0,Y 505.815,Z 358.22,A -85,B 0,C 180,E1 24237.425,E2 24237.425} C_VEL
LIN {X 0,Y 505.81,Z 358.209,A -85,B 0,C 180,E1 24233.906,E2 24233.906} C_VEL
LIN {X 0,Y 505.865,Z 358.204,A -85,B 0,C 180,E1 24230.599,E2 24230.599} C_VEL
LIN {X 0,Y 505.803,Z 358.216,A -85,B 0,C 180,E1 24227.249,E2 24227.249} C_VEL
LIN {X 0,Y 505.813,Z 358.227,A -85,B 0,C 180,E1 24223.722,E2 24223.722} C_VEL
LIN {X 0,Y 505.848,Z 358.212,A -85,B 0,C 180,E1 24220.362,E2 24220.362} C_VEL
LIN {X 0,Y 505.791,Z 358.217,A -85,B 0,C 180,E1 24217.04,E2 24217.04} C_VEL
LIN {X 0,Y 505.874,Z 358.565,A -85,B 0,C 180,E1 24216.469,E2 24216.469} C_VEL
LIN {X 0,Y 506.305,Z 360.03,A -85,B 0,C 180,E1 24216.15,E2 24216.15} C_VEL
LIN {X 0,Y 508.039,Z 362.829,A -85,B 0,C 180,E1 24215.591,E2 24215.591} C_VEL
LIN {X 0,Y 511.249,Z 365.265,A -85,B 0,C 180,E1 24214.698,E2 24214.698} C_VEL
LIN {X 0,Y 513.492,Z 368.958,A -85,B 0,C 180,E1 24214.02,E2 24214.02} C_VEL
LIN {X 0,Y 516.652,Z 371.682,A -85,B 0,C 180,E1 24213.187,E2 24213.187} C_VEL
LIN {X 0,Y 519.408,Z 375.62,A -85,B 0,C 180,E1 24212.415,E2 24212.415} C_VEL
LIN {X 0,Y 521.799,Z 377.844,A -85,B 0,C 180,E1 24211.812,E2 24211.812} C_VEL
LIN {X 0,Y 525.024,Z 382.074,A -85,B 0,C 180,E1 24210.988,E2 24210.988} C_VEL
LIN {X 0,Y 526.967,Z 384.018,A -85,B 0,C 180,E1 24210.523,E2 24210.523} C_VEL
LIN {X 0,Y 530.528,Z 388.511,A -85,B 0,C 180,E1 24209.649,E2 24209.649} C_VEL
LIN {X 0,Y 532.49,Z 390.669,A -85,B 0,C 180,E1 24209.193,E2 24209.193} C_VEL
LIN {X 0,Y 537.612,Z 396.917,A -85,B 0,C 180,E1 24208.028,E2 24208.028} C_VEL
LIN {X 0,Y 542.2,Z 402.711,A -85,B 0,C 180,E1 24207.014,E2 24207.014} C_VEL
LIN {X 0,Y 550.162,Z 412.354,A -85,B 0,C 180,E1 24205.361,E2 24205.361} C_VEL
LIN {X 0,Y 565.984,Z 432.749,A -85,B 0,C 180,E1 24202.346,E2 24202.346} C_VEL
LIN {X 0,Y 577.65,Z 448.551,A -85,B 0,C 180,E1 24200.32,E2 24200.32} C_VEL
LIN {X 0,Y 578.539,Z 451.328,A -85,B 0,C 180,E1 24200.136,E2 24200.136} C_VEL
LIN {X 0,Y 578.535,Z 455.563,A -85,B 0,C 180,E1 24200.042,E2 24200.042} C_VEL
LIN {X 0,Y 577.2,Z 462.51,A -85,B 0,C 180,E1 24200.067,E2 24200.067} C_VEL
LIN {X 0,Y 575.503,Z 470.682,A -85,B 0,C 180,E1 24200.109,E2 24200.109} C_VEL
LIN {X 0,Y 575.359,Z 472.329,A -85,B 0,C 180,E1 24200.091,E2 24200.091} C_VEL
LIN {X 0,Y 565.416,Z 677.879,A -85,B 0,C 180,E1 24196.914,E2 24196.914} C_VEL
LIN {X 0,Y 561.307,Z 767.614,A -85,B 0,C 180,E1 24195.532,E2 24195.532} C_VEL
LIN {X 0,Y 559.085,Z 796.336,A -85,B 0,C 180,E1 24194.929,E2 24194.929} C_VEL
LIN {X 0,Y 556.594,Z 820.179,A -85,B 0,C 180,E1 24194.261,E2 24194.261} C_VEL
LIN {X 0,Y 553.967,Z 841.316,A -85,B 0,C 180,E1 24193.538,E2 24193.538} C_VEL
LIN {X 0,Y 550.93,Z 862.541,A -85,B 0,C 180,E1 24192.679,E2 24192.679} C_VEL
LIN {X 0,Y 546.748,Z 888.176,A -85,B 0,C 180,E1 24191.446,E2 24191.446} C_VEL
LIN {X 0,Y 542.605,Z 910.273,A -85,B 0,C 180,E1 24190.18,E2 24190.18} C_VEL
LIN {X 0,Y 538.851,Z 928.819,A -85,B 0,C 180,E1 24188.966,E2 24188.966} C_VEL
LIN {X 0,Y 535.145,Z 945.87,A -85,B 0,C 180,E1 24187.71,E2 24187.71} C_VEL
LIN {X 0,Y 531.055,Z 963.639,A -85,B 0,C 180,E1 24186.239,E2 24186.239} C_VEL
LIN {X 0,Y 526.086,Z 984.482,A -85,B 0,C 180,E1 24184.277,E2 24184.277} C_VEL
LIN {X 0,Y 521.288,Z 1003.284,A -85,B 0,C 180,E1 24182.219,E2 24182.219} C_VEL
LIN {X 0,Y 517.501,Z 1018.021,A -85,B 0,C 180,E1 24180.398,E2 24180.398} C_VEL
LIN {X 0,Y 513.585,Z 1033.175,A -85,B 0,C 180,E1 24178.298,E2 24178.298} C_VEL
LIN {X 0,Y 509.192,Z 1050.359,A -85,B 0,C 180,E1 24175.561,E2 24175.561} C_VEL
LIN {X 0,Y 505.623,Z 1064.597,A -85,B 0,C 180,E1 24172.905,E2 24172.905} C_VEL
LIN {X 0,Y 502.576,Z 1077.677,A -85,B 0,C 180,E1 24170.078,E2 24170.078} C_VEL
LIN {X 0,Y 499.612,Z 1093.123,A -85,B 0,C 180,E1 24166.26,E2 24166.26} C_VEL
LIN {X 0,Y 498.113,Z 1103.208,A -85,B 0,C 180,E1 24163.355,E2 24163.355} C_VEL
LIN {X 0,Y 497.06,Z 1111.823,A -85,B 0,C 180,E1 24160.372,E2 24160.372} C_VEL
LIN {X 0,Y 496.386,Z 1119.1,A -85,B 0,C 180,E1 24157.283,E2 24157.283} C_VEL
LIN {X 0,Y 496.086,Z 1124.673,A -85,B 0,C 180,E1 24154.273,E2 24154.273} C_VEL
LIN {X 0,Y 495.95,Z 1128.582,A -85,B 0,C 180,E1 24151.261,E2 24151.261} C_VEL
LIN {X 0,Y 495.919,Z 1131.024,A -85,B 0,C 180,E1 24148.282,E2 24148.282} C_VEL
LIN {X 0,Y 495.902,Z 1131.933,A -85,B 0,C 180,E1 24145.406,E2 24145.406} C_VEL
LIN {X 0,Y 495.874,Z 1131.449,A -85,B 0,C 180,E1 24142.527,E2 24142.527} C_VEL
LIN {X 0,Y 495.934,Z 1129.724,A -85,B 0,C 180,E1 24139.799,E2 24139.799} C_VEL
LIN {X 0,Y 495.985,Z 1126.435,A -85,B 0,C 180,E1 24136.876,E2 24136.876} C_VEL
LIN {X 0,Y 496.194,Z 1121.856,A -85,B 0,C 180,E1 24133.994,E2 24133.994} C_VEL
LIN {X 0,Y 496.707,Z 1115.533,A -85,B 0,C 180,E1 24131.025,E2 24131.025} C_VEL
LIN {X 0,Y 497.609,Z 1107.128,A -85,B 0,C 180,E1 24127.853,E2 24127.853} C_VEL
LIN {X 0,Y 498.958,Z 1097.448,A -85,B 0,C 180,E1 24124.828,E2 24124.828} C_VEL
LIN {X 0,Y 500.878,Z 1085.999,A -85,B 0,C 180,E1 24121.83,E2 24121.83} C_VEL
LIN {X 0,Y 504.422,Z 1070.864,A -85,B 0,C 180,E1 24118.183,E2 24118.183} C_VEL
LIN {X 0,Y 507.997,Z 1057.036,A -85,B 0,C 180,E1 24115.371,E2 24115.371} C_VEL
LIN {X 0,Y 511.395,Z 1044.44,A -85,B 0,C 180,E1 24113.15,E2 24113.15} C_VEL
LIN {X 0,Y 515.253,Z 1030.354,A -85,B 0,C 180,E1 24110.956,E2 24110.956} C_VEL
LIN {X 0,Y 519.996,Z 1012.694,A -85,B 0,C 180,E1 24108.577,E2 24108.577} C_VEL
LIN {X 0,Y 524.011,Z 997.237,A -85,B 0,C 180,E1 24106.763,E2 24106.763} C_VEL
LIN {X 0,Y 527.963,Z 981.587,A -85,B 0,C 180,E1 24105.13,E2 24105.13} C_VEL
LIN {X 0,Y 532.429,Z 962.966,A -85,B 0,C 180,E1 24103.414,E2 24103.414} C_VEL
LIN {X 0,Y 537.087,Z 941.536,A -85,B 0,C 180,E1 24101.718,E2 24101.718} C_VEL
LIN {X 0,Y 540.786,Z 923.066,A -85,B 0,C 180,E1 24100.448,E2 24100.448} C_VEL
LIN {X 0,Y 544.126,Z 904.688,A -85,B 0,C 180,E1 24099.34,E2 24099.34} C_VEL
LIN {X 0,Y 547.684,Z 882.783,A -85,B 0,C 180,E1 24098.19,E2 24098.19} C_VEL
LIN {X 0,Y 550.85,Z 858.849,A -85,B 0,C 180,E1 24097.142,E2 24097.142} C_VEL
LIN {X 0,Y 553.257,Z 837.407,A -85,B 0,C 180,E1 24096.36,E2 24096.36} C_VEL
LIN {X 0,Y 555.341,Z 814.693,A -85,B 0,C 180,E1 24095.674,E2 24095.674} C_VEL
LIN {X 0,Y 557.122,Z 787.529,A -85,B 0,C 180,E1 24095.043,E2 24095.043} C_VEL
LIN {X 0,Y 563.331,Z 679.437,A -85,B 0,C 180,E1 24093.213,E2 24093.213} C_VEL
LIN {X 0,Y 569.114,Z 608.161,A -85,B 0,C 180,E1 24091.924,E2 24091.924} C_VEL
LIN {X 0,Y 576.42,Z 540.981,A -85,B 0,C 180,E1 24090.635,E2 24090.635} C_VEL
LIN {X 0,Y 584.867,Z 481.204,A -85,B 0,C 180,E1 24089.447,E2 24089.447} C_VEL
LIN {X 0,Y 587.394,Z 465.715,A -85,B 0,C 180,E1 24089.115,E2 24089.115} C_VEL
LIN {X 0,Y 585.503,Z 474.1,A -85,B 0,C 180,E1 24088.132,E2 24088.132} C_VEL
LIN {X 0,Y 583.084,Z 492.343,A -85,B 0,C 180,E1 24087.188,E2 24087.188} C_VEL
LIN {X 0,Y 582.7,Z 496.05,A -85,B 0,C 180,E1 24087.014,E2 24087.014} C_VEL
LIN {X 0,Y 574.716,Z 556.729,A -85,B 0,C 180,E1 24085.785,E2 24085.785} C_VEL
LIN {X 0,Y 568.032,Z 622.862,A -85,B 0,C 180,E1 24084.5,E2 24084.5} C_VEL
LIN {X 0,Y 562.367,Z 697.717,A -85,B 0,C 180,E1 24083.136,E2 24083.136} C_VEL
LIN {X 0,Y 557.957,Z 777.345,A -85,B 0,C 180,E1 24081.79,E2 24081.79} C_VEL
LIN {X 0,Y 553.332,Z 882.721,A -85,B 0,C 180,E1 24080.107,E2 24080.107} C_VEL
LIN {X 0,Y 551.004,Z 911.586,A -85,B 0,C 180,E1 24079.511,E2 24079.511} C_VEL
LIN {X 0,Y 548.434,Z 936.923,A -85,B 0,C 180,E1 24078.868,E2 24078.868} C_VEL
LIN {X 0,Y 544.765,Z 968.575,A -85,B 0,C 180,E1 24077.86,E2 24077.86} C_VEL
LIN {X 0,Y 541.559,Z 993.852,A -85,B 0,C 180,E1 24076.869,E2 24076.869} C_VEL
LIN {X 0,Y 538.456,Z 1016.508,A -85,B 0,C 180,E1 24075.837,E2 24075.837} C_VEL
LIN {X 0,Y 534.445,Z 1044.109,A -85,B 0,C 180,E1 24074.383,E2 24074.383} C_VEL
LIN {X 0,Y 530.554,Z 1068.774,A -85,B 0,C 180,E1 24072.852,E2 24072.852} C_VEL
LIN {X 0,Y 527.359,Z 1088.113,A -85,B 0,C 180,E1 24071.502,E2 24071.502} C_VEL
LIN {X 0,Y 524.22,Z 1106.359,A -85,B 0,C 180,E1 24070.085,E2 24070.085} C_VEL
LIN {X 0,Y 521.008,Z 1124.547,A -85,B 0,C 180,E1 24068.517,E2 24068.517} C_VEL
LIN {X 0,Y 517.849,Z 1142.125,A -85,B 0,C 180,E1 24066.835,E2 24066.835} C_VEL
LIN {X 0,Y 514.543,Z 1160.181,A -85,B 0,C 180,E1 24064.909,E2 24064.909} C_VEL
LIN {X 0,Y 510.753,Z 1180.596,A -85,B 0,C 180,E1 24062.439,E2 24062.439} C_VEL
LIN {X 0,Y 507.907,Z 1196.388,A -85,B 0,C 180,E1 24060.263,E2 24060.263} C_VEL
LIN {X 0,Y 505.512,Z 1209.768,A -85,B 0,C 180,E1 24058.212,E2 24058.212} C_VEL
LIN {X 0,Y 503.364,Z 1222.014,A -85,B 0,C 180,E1 24056.121,E2 24056.121} C_VEL
LIN {X 0,Y 501.952,Z 1230.189,A -85,B 0,C 180,E1 24054.477,E2 24054.477} C_VEL
LIN {X 0,Y 499.961,Z 1241.053,A -85,B 0,C 180,E1 24051.838,E2 24051.838} C_VEL
LIN {X 0,Y 498.57,Z 1249.695,A -85,B 0,C 180,E1 24049.445,E2 24049.445} C_VEL
LIN {X 0,Y 497.544,Z 1257.559,A -85,B 0,C 180,E1 24046.942,E2 24046.942} C_VEL
LIN {X 0,Y 496.675,Z 1265.759,A -85,B 0,C 180,E1 24043.861,E2 24043.861} C_VEL
LIN {X 0,Y 496.212,Z 1272.067,A -85,B 0,C 180,E1 24040.801,E2 24040.801} C_VEL
LIN {X 0,Y 495.998,Z 1276.256,A -85,B 0,C 180,E1 24038.182,E2 24038.182} C_VEL
LIN {X 0,Y 495.939,Z 1279.081,A -85,B 0,C 180,E1 24035.786,E2 24035.786} C_VEL
LIN {X 0,Y 495.912,Z 1280.946,A -85,B 0,C 180,E1 24033.352,E2 24033.352} C_VEL
LIN {X 0,Y 495.877,Z 1281.803,A -85,B 0,C 180,E1 24031.04,E2 24031.04} C_VEL
LIN {X 0,Y 495.892,Z 1281.757,A -85,B 0,C 180,E1 24028.729,E2 24028.729} C_VEL
LIN {X 0,Y 495.913,Z 1280.809,A -85,B 0,C 180,E1 24026.416,E2 24026.416} C_VEL
LIN {X 0,Y 495.946,Z 1278.852,A -85,B 0,C 180,E1 24023.982,E2 24023.982} C_VEL
LIN {X 0,Y 496.045,Z 1275.552,A -85,B 0,C 180,E1 24021.305,E2 24021.305} C_VEL
LIN {X 0,Y 496.339,Z 1270.086,A -85,B 0,C 180,E1 24018.142,E2 24018.142} C_VEL
LIN {X 0,Y 496.844,Z 1263.649,A -85,B 0,C 180,E1 24015.311,E2 24015.311} C_VEL
LIN {X 0,Y 497.622,Z 1256.852,A -85,B 0,C 180,E1 24012.82,E2 24012.82} C_VEL
LIN {X 0,Y 498.629,Z 1249.289,A -85,B 0,C 180,E1 24010.435,E2 24010.435} C_VEL
LIN {X 0,Y 500.04,Z 1240.598,A -85,B 0,C 180,E1 24008.042,E2 24008.042} C_VEL
LIN {X 0,Y 502.162,Z 1229.149,A -85,B 0,C 180,E1 24005.283,E2 24005.283} C_VEL
LIN {X 0,Y 504.739,Z 1214.659,A -85,B 0,C 180,E1 24002.512,E2 24002.512} C_VEL
LIN {X 0,Y 507.515,Z 1200.188,A -85,B 0,C 180,E1 24000.098,E2 24000.098} C_VEL
LIN {X 0,Y 510.24,Z 1186.565,A -85,B 0,C 180,E1 23998.052,E2 23998.052} C_VEL
LIN {X 0,Y 513.451,Z 1171.094,A -85,B 0,C 180,E1 23995.953,E2 23995.953} C_VEL
LIN {X 0,Y 517.786,Z 1150.859,A -85,B 0,C 180,E1 23993.504,E2 23993.504} C_VEL
LIN {X 0,Y 522.067,Z 1130.846,A -85,B 0,C 180,E1 23991.391,E2 23991.391} C_VEL
LIN {X 0,Y 525.845,Z 1113.211,A -85,B 0,C 180,E1 23989.722,E2 23989.722} C_VEL
LIN {X 0,Y 529.817,Z 1094.42,A -85,B 0,C 180,E1 23988.124,E2 23988.124} C_VEL
LIN {X 0,Y 534.665,Z 1071.083,A -85,B 0,C 180,E1 23986.364,E2 23986.364} C_VEL
LIN {X 0,Y 539.347,Z 1046.565,A -85,B 0,C 180,E1 23984.788,E2 23984.788} C_VEL
LIN {X 0,Y 543.059,Z 1026.287,A -85,B 0,C 180,E1 23983.648,E2 23983.648} C_VEL
LIN {X 0,Y 546.48,Z 1006.072,A -85,B 0,C 180,E1 23982.648,E2 23982.648} C_VEL
LIN {X 0,Y 550.339,Z 981.715,A -85,B 0,C 180,E1 23981.615,E2 23981.615} C_VEL
LIN {X 0,Y 554.152,Z 953.843,A -85,B 0,C 180,E1 23980.656,E2 23980.656} C_VEL
LIN {X 0,Y 556.809,Z 931.369,A -85,B 0,C 180,E1 23980.035,E2 23980.035} C_VEL
LIN {X 0,Y 559.023,Z 909.053,A -85,B 0,C 180,E1 23979.543,E2 23979.543} C_VEL
LIN {X 0,Y 560.828,Z 882.125,A -85,B 0,C 180,E1 23979.07,E2 23979.07} C_VEL
LIN {X 0,Y 569.772,Z 677.215,A -85,B 0,C 180,E1 23975.941,E2 23975.941} C_VEL
LIN {X 0,Y 579.051,Z 494.101,A -85,B 0,C 180,E1 23973.059,E2 23973.059} C_VEL
LIN {X 0,Y 576.756,Z 479.323,A -85,B 0,C 180,E1 23972.391,E2 23972.391} C_VEL
LIN {X 0,Y 564.953,Z 461.052,A -85,B 0,C 180,E1 23970.204,E2 23970.204} C_VEL
LIN {X 0,Y 553.358,Z 443.821,A -85,B 0,C 180,E1 23967.875,E2 23967.875} C_VEL
LIN {X 0,Y 540.796,Z 425.979,A -85,B 0,C 180,E1 23965.137,E2 23965.137} C_VEL
LIN {X 0,Y 529.786,Z 410.953,A -85,B 0,C 180,E1 23962.499,E2 23962.499} C_VEL
LIN {X 0,Y 521.537,Z 399.824,A -85,B 0,C 180,E1 23960.305,E2 23960.305} C_VEL
LIN {X 0,Y 518.732,Z 395.027,A -85,B 0,C 180,E1 23959.128,E2 23959.128} C_VEL
LIN {X 0,Y 515.903,Z 390.056,A -85,B 0,C 180,E1 23957.832,E2 23957.832} C_VEL
LIN {X 0,Y 513.381,Z 385.571,A -85,B 0,C 180,E1 23956.637,E2 23956.637} C_VEL
LIN {X 0,Y 510.923,Z 381.241,A -85,B 0,C 180,E1 23955.436,E2 23955.436} C_VEL
LIN {X 0,Y 508.054,Z 376.502,A -85,B 0,C 180,E1 23954.009,E2 23954.009} C_VEL
LIN {X 0,Y 504.849,Z 371.235,A -85,B 0,C 180,E1 23952.351,E2 23952.351} C_VEL
LIN {X 0,Y 503.792,Z 369.578,A -85,B 0,C 180,E1 23951.796,E2 23951.796} C_VEL
LIN {X 0,Y 501.572,Z 365.944,A -85,B 0,C 180,E1 23950.568,E2 23950.568} C_VEL
LIN {X 0,Y 500.851,Z 364.533,A -85,B 0,C 180,E1 23950.118,E2 23950.118} C_VEL
LIN {X 0,Y 498.51,Z 361.339,A -85,B 0,C 180,E1 23948.885,E2 23948.885} C_VEL
LIN {X 0,Y 497.938,Z 359.393,A -85,B 0,C 180,E1 23948.197,E2 23948.197} C_VEL
LIN {X 0,Y 497.927,Z 359.185,A -85,B 0,C 180,E1 23944.723,E2 23944.723} C_VEL
LIN {X 0,Y 497.918,Z 359.186,A -85,B 0,C 180,E1 23941.151,E2 23941.151} C_VEL
LIN {X 0,Y 497.9,Z 359.21,A -85,B 0,C 180,E1 23937.698,E2 23937.698} C_VEL
LIN {X 0,Y 497.926,Z 359.209,A -85,B 0,C 180,E1 23934.122,E2 23934.122} C_VEL
LIN {X 0,Y 497.928,Z 359.205,A -85,B 0,C 180,E1 23930.639,E2 23930.639} C_VEL
LIN {X 0,Y 497.895,Z 359.207,A -85,B 0,C 180,E1 23927.12,E2 23927.12} C_VEL
LIN {X 0,Y 497.913,Z 359.201,A -85,B 0,C 180,E1 23923.671,E2 23923.671} C_VEL
LIN {X 0,Y 497.932,Z 359.195,A -85,B 0,C 180,E1 23920.162,E2 23920.162} C_VEL
LIN {X 0,Y 497.891,Z 359.196,A -85,B 0,C 180,E1 23916.695,E2 23916.695} C_VEL
LIN {X 0,Y 497.893,Z 359.2,A -85,B 0,C 180,E1 23913.081,E2 23913.081} C_VEL
LIN {X 0,Y 497.936,Z 359.196,A -85,B 0,C 180,E1 23909.6,E2 23909.6} C_VEL
LIN {X 0,Y 497.907,Z 359.208,A -85,B 0,C 180,E1 23906.063,E2 23906.063} C_VEL
LIN {X 0,Y 497.882,Z 359.213,A -85,B 0,C 180,E1 23902.518,E2 23902.518} C_VEL
LIN {X 0,Y 497.92,Z 359.206,A -85,B 0,C 180,E1 23899.106,E2 23899.106} C_VEL
LIN {X 0,Y 497.91,Z 359.204,A -85,B 0,C 180,E1 23895.635,E2 23895.635} C_VEL
LIN {X 0,Y 497.875,Z 359.202,A -85,B 0,C 180,E1 23892.177,E2 23892.177} C_VEL
LIN {X 0,Y 497.913,Z 359.196,A -85,B 0,C 180,E1 23888.795,E2 23888.795} C_VEL
LIN {X 0,Y 497.903,Z 359.196,A -85,B 0,C 180,E1 23885.335,E2 23885.335} C_VEL
LIN {X 0,Y 497.87,Z 359.202,A -85,B 0,C 180,E1 23881.839,E2 23881.839} C_VEL
LIN {X 0,Y 497.902,Z 359.201,A -85,B 0,C 180,E1 23878.406,E2 23878.406} C_VEL
LIN {X 0,Y 497.906,Z 359.207,A -85,B 0,C 180,E1 23874.943,E2 23874.943} C_VEL
LIN {X 0,Y 497.865,Z 359.208,A -85,B 0,C 180,E1 23871.563,E2 23871.563} C_VEL
LIN {X 0,Y 497.898,Z 359.198,A -85,B 0,C 180,E1 23868.136,E2 23868.136} C_VEL
LIN {X 0,Y 497.886,Z 359.2,A -85,B 0,C 180,E1 23864.776,E2 23864.776} C_VEL
LIN {X 0,Y 497.859,Z 359.215,A -85,B 0,C 180,E1 23861.351,E2 23861.351} C_VEL
LIN {X 0,Y 497.905,Z 359.426,A -85,B 0,C 180,E1 23858.662,E2 23858.662} C_VEL
LIN {X 0,Y 498.261,Z 360.733,A -85,B 0,C 180,E1 23858.265,E2 23858.265} C_VEL
LIN {X 0,Y 499.993,Z 363.702,A -85,B 0,C 180,E1 23857.642,E2 23857.642} C_VEL
LIN {X 0,Y 503.432,Z 366.275,A -85,B 0,C 180,E1 23856.615,E2 23856.615} C_VEL
LIN {X 0,Y 505.424,Z 369.742,A -85,B 0,C 180,E1 23855.962,E2 23855.962} C_VEL
LIN {X 0,Y 508.867,Z 372.678,A -85,B 0,C 180,E1 23854.978,E2 23854.978} C_VEL
LIN {X 0,Y 511.542,Z 376.657,A -85,B 0,C 180,E1 23854.175,E2 23854.175} C_VEL
LIN {X 0,Y 514.251,Z 379.074,A -85,B 0,C 180,E1 23853.456,E2 23853.456} C_VEL
LIN {X 0,Y 517.464,Z 383.322,A -85,B 0,C 180,E1 23852.562,E2 23852.562} C_VEL
LIN {X 0,Y 519.475,Z 385.405,A -85,B 0,C 180,E1 23852.041,E2 23852.041} C_VEL
LIN {X 0,Y 523.047,Z 389.774,A -85,B 0,C 180,E1 23851.128,E2 23851.128} C_VEL
LIN {X 0,Y 524.754,Z 391.772,A -85,B 0,C 180,E1 23850.71,E2 23850.71} C_VEL
LIN {X 0,Y 528.703,Z 396.343,A -85,B 0,C 180,E1 23849.754,E2 23849.754} C_VEL
LIN {X 0,Y 535.196,Z 404.384,A -85,B 0,C 180,E1 23848.242,E2 23848.242} C_VEL
LIN {X 0,Y 539.869,Z 410.269,A -85,B 0,C 180,E1 23847.213,E2 23847.213} C_VEL
LIN {X 0,Y 547.282,Z 419.31,A -85,B 0,C 180,E1 23845.652,E2 23845.652} C_VEL
LIN {X 0,Y 562.744,Z 439.351,A -85,B 0,C 180,E1 23842.667,E2 23842.667} C_VEL
LIN {X 0,Y 576.124,Z 457.739,A -85,B 0,C 180,E1 23840.321,E2 23840.321} C_VEL
LIN {X 0,Y 575.359,Z 472.329,A -85,B 0,C 180,E1 23840.091,E2 23840.091} C_VEL
LIN {X 0,Y 574.346,Z 480.02,A -85,B 0,C 180,E1 23840.051,E2 23840.051} C_VEL
LIN {X 0,Y 569.516,Z 500.634,A -85,B 0,C 180,E1 23840.231,E2 23840.231} C_VEL
LIN {X 0,Y 568.713,Z 507.23,A -85,B 0,C 180,E1 23840.188,E2 23840.188} C_VEL
LIN {X 0,Y 558.896,Z 707.593,A -85,B 0,C 180,E1 23837.085,E2 23837.085} C_VEL
LIN {X 0,Y 555.702,Z 772.042,A -85,B 0,C 180,E1 23836.07,E2 23836.07} C_VEL
LIN {X 0,Y 553.372,Z 799.671,A -85,B 0,C 180,E1 23835.46,E2 23835.46} C_VEL
LIN {X 0,Y 550.969,Z 821.988,A -85,B 0,C 180,E1 23834.824,E2 23834.824} C_VEL
LIN {X 0,Y 548.386,Z 842.22,A -85,B 0,C 180,E1 23834.128,E2 23834.128} C_VEL
LIN {X 0,Y 545.273,Z 863.324,A -85,B 0,C 180,E1 23833.268,E2 23833.268} C_VEL
LIN {X 0,Y 541.183,Z 887.906,A -85,B 0,C 180,E1 23832.086,E2 23832.086} C_VEL
LIN {X 0,Y 536.66,Z 911.249,A -85,B 0,C 180,E1 23830.745,E2 23830.745} C_VEL
LIN {X 0,Y 532.95,Z 929.027,A -85,B 0,C 180,E1 23829.577,E2 23829.577} C_VEL
LIN {X 0,Y 529.138,Z 946.073,A -85,B 0,C 180,E1 23828.32,E2 23828.32} C_VEL
LIN {X 0,Y 525.063,Z 963.304,A -85,B 0,C 180,E1 23826.896,E2 23826.896} C_VEL
LIN {X 0,Y 520.702,Z 980.926,A -85,B 0,C 180,E1 23825.253,E2 23825.253} C_VEL
LIN {X 0,Y 515.125,Z 1002.54,A -85,B 0,C 180,E1 23822.93,E2 23822.93} C_VEL
LIN {X 0,Y 510.975,Z 1018.086,A -85,B 0,C 180,E1 23821.01,E2 23821.01} C_VEL
LIN {X 0,Y 507.259,Z 1031.865,A -85,B 0,C 180,E1 23819.104,E2 23819.104} C_VEL
LIN {X 0,Y 503.47,Z 1046.059,A -85,B 0,C 180,E1 23816.897,E2 23816.897} C_VEL
LIN {X 0,Y 499.258,Z 1062.147,A -85,B 0,C 180,E1 23814.01,E2 23814.01} C_VEL
LIN {X 0,Y 496.163,Z 1074.426,A -85,B 0,C 180,E1 23811.437,E2 23811.437} C_VEL
LIN {X 0,Y 493.347,Z 1086.552,A -85,B 0,C 180,E1 23808.491,E2 23808.491} C_VEL
LIN {X 0,Y 490.661,Z 1100.677,A -85,B 0,C 180,E1 23804.437,E2 23804.437} C_VEL
LIN {X 0,Y 489.311,Z 1110.202,A -85,B 0,C 180,E1 23801.238,E2 23801.238} C_VEL
LIN {X 0,Y 488.588,Z 1117.38,A -85,B 0,C 180,E1 23798.323,E2 23798.323} C_VEL
LIN {X 0,Y 488.165,Z 1123.223,A -85,B 0,C 180,E1 23795.283,E2 23795.283} C_VEL
LIN {X 0,Y 487.965,Z 1127.534,A -85,B 0,C 180,E1 23792.332,E2 23792.332} C_VEL
LIN {X 0,Y 487.924,Z 1130.175,A -85,B 0,C 180,E1 23789.596,E2 23789.596} C_VEL
LIN {X 0,Y 487.88,Z 1131.737,A -85,B 0,C 180,E1 23786.669,E2 23786.669} C_VEL
LIN {X 0,Y 487.899,Z 1131.848,A -85,B 0,C 180,E1 23783.935,E2 23783.935} C_VEL
LIN {X 0,Y 487.918,Z 1130.593,A -85,B 0,C 180,E1 23780.858,E2 23780.858} C_VEL
LIN {X 0,Y 487.965,Z 1128.057,A -85,B 0,C 180,E1 23778.053,E2 23778.053} C_VEL
LIN {X 0,Y 488.148,Z 1123.777,A -85,B 0,C 180,E1 23774.957,E2 23774.957} C_VEL
LIN {X 0,Y 488.538,Z 1117.868,A -85,B 0,C 180,E1 23771.81,E2 23771.81} C_VEL
LIN {X 0,Y 489.228,Z 1110.91,A -85,B 0,C 180,E1 23768.936,E2 23768.936} C_VEL
LIN {X 0,Y 490.472,Z 1101.829,A -85,B 0,C 180,E1 23765.827,E2 23765.827} C_VEL
LIN {X 0,Y 493.563,Z 1086.466,A -85,B 0,C 180,E1 23761.277,E2 23761.277} C_VEL
LIN {X 0,Y 496.347,Z 1075.355,A -85,B 0,C 180,E1 23758.499,E2 23758.499} C_VEL
LIN {X 0,Y 499.97,Z 1062.141,A -85,B 0,C 180,E1 23755.642,E2 23755.642} C_VEL
LIN {X 0,Y 503.881,Z 1047.948,A -85,B 0,C 180,E1 23753.047,E2 23753.047} C_VEL
LIN {X 0,Y 507.413,Z 1035.499,A -85,B 0,C 180,E1 23751.044,E2 23751.044} C_VEL
LIN {X 0,Y 511.08,Z 1022.465,A -85,B 0,C 180,E1 23749.175,E2 23749.175} C_VEL
LIN {X 0,Y 515.852,Z 1005.386,A -85,B 0,C 180,E1 23747.006,E2 23747.006} C_VEL
LIN {X 0,Y 520.73,Z 986.699,A -85,B 0,C 180,E1 23744.976,E2 23744.976} C_VEL
LIN {X 0,Y 524.712,Z 970.784,A -85,B 0,C 180,E1 23743.448,E2 23743.448} C_VEL
LIN {X 0,Y 528.744,Z 953.649,A -85,B 0,C 180,E1 23741.99,E2 23741.99} C_VEL
LIN {X 0,Y 533.426,Z 932.186,A -85,B 0,C 180,E1 23740.395,E2 23740.395} C_VEL
LIN {X 0,Y 537.419,Z 911.258,A -85,B 0,C 180,E1 23739.07,E2 23739.07} C_VEL
LIN {X 0,Y 540.704,Z 892.012,A -85,B 0,C 180,E1 23738.008,E2 23738.008} C_VEL
LIN {X 0,Y 544.055,Z 869.804,A -85,B 0,C 180,E1 23736.954,E2 23736.954} C_VEL
LIN {X 0,Y 547.195,Z 844.132,A -85,B 0,C 180,E1 23735.953,E2 23735.953} C_VEL
LIN {X 0,Y 549.283,Z 823.344,A -85,B 0,C 180,E1 23735.286,E2 23735.286} C_VEL
LIN {X 0,Y 551.267,Z 798.505,A -85,B 0,C 180,E1 23734.641,E2 23734.641} C_VEL
LIN {X 0,Y 553.231,Z 763.117,A -85,B 0,C 180,E1 23733.977,E2 23733.977} C_VEL
LIN {X 0,Y 558.434,Z 685.969,A -85,B 0,C 180,E1 23732.642,E2 23732.642} C_VEL
LIN {X 0,Y 564.817,Z 616.148,A -85,B 0,C 180,E1 23731.342,E2 23731.342} C_VEL
LIN {X 0,Y 572.742,Z 551.832,A -85,B 0,C 180,E1 23730.075,E2 23730.075} C_VEL
LIN {X 0,Y 581.863,Z 493.791,A -85,B 0,C 180,E1 23728.906,E2 23728.906} C_VEL
LIN {X 0,Y 584.06,Z 481.543,A -85,B 0,C 180,E1 23728.643,E2 23728.643} C_VEL
LIN {X 0,Y 581.078,Z 498.564,A -85,B 0,C 180,E1 23727.754,E2 23727.754} C_VEL
LIN {X 0,Y 572.04,Z 557.756,A -85,B 0,C 180,E1 23726.531,E2 23726.531} C_VEL
LIN {X 0,Y 564.613,Z 620.157,A -85,B 0,C 180,E1 23725.277,E2 23725.277} C_VEL
LIN {X 0,Y 558.561,Z 687.033,A -85,B 0,C 180,E1 23724.005,E2 23724.005} C_VEL
LIN {X 0,Y 553.575,Z 760.62,A -85,B 0,C 180,E1 23722.694,E2 23722.694} C_VEL
LIN {X 0,Y 547.504,Z 880.965,A -85,B 0,C 180,E1 23720.7,E2 23720.7} C_VEL
LIN {X 0,Y 545.095,Z 909.28,A -85,B 0,C 180,E1 23720.103,E2 23720.103} C_VEL
LIN {X 0,Y 542.183,Z 936.502,A -85,B 0,C 180,E1 23719.402,E2 23719.402} C_VEL
LIN {X 0,Y 538.427,Z 966.977,A -85,B 0,C 180,E1 23718.413,E2 23718.413} C_VEL
LIN {X 0,Y 535.081,Z 992.294,A -85,B 0,C 180,E1 23717.412,E2 23717.412} C_VEL
LIN {X 0,Y 531.35,Z 1018.633,A -85,B 0,C 180,E1 23716.191,E2 23716.191} C_VEL
LIN {X 0,Y 527.027,Z 1046.506,A -85,B 0,C 180,E1 23714.661,E2 23714.661} C_VEL
LIN {X 0,Y 523.634,Z 1067.314,A -85,B 0,C 180,E1 23713.351,E2 23713.351} C_VEL
LIN {X 0,Y 520.436,Z 1086.024,A -85,B 0,C 180,E1 23712.032,E2 23712.032} C_VEL
LIN {X 0,Y 517.14,Z 1104.613,A -85,B 0,C 180,E1 23710.58,E2 23710.58} C_VEL
LIN {X 0,Y 513.81,Z 1122.784,A -85,B 0,C 180,E1 23709,E2 23709} C_VEL
LIN {X 0,Y 510.623,Z 1139.974,A -85,B 0,C 180,E1 23707.343,E2 23707.343} C_VEL
LIN {X 0,Y 507.257,Z 1157.932,A -85,B 0,C 180,E1 23705.416,E2 23705.416} C_VEL
LIN {X 0,Y 503.242,Z 1178.97,A -85,B 0,C 180,E1 23702.848,E2 23702.848} C_VEL
LIN {X 0,Y 500.422,Z 1193.997,A -85,B 0,C 180,E1 23700.764,E2 23700.764} C_VEL
LIN {X 0,Y 498.077,Z 1206.773,A -85,B 0,C 180,E1 23698.803,E2 23698.803} C_VEL
LIN {X 0,Y 495.789,Z 1219.654,A -85,B 0,C 180,E1 23696.597,E2 23696.597} C_VEL
LIN {X 0,Y 493.846,Z 1231.143,A -85,B 0,C 180,E1 23694.395,E2 23694.395} C_VEL
LIN {X 0,Y 492.56,Z 1239.074,A -85,B 0,C 180,E1 23692.687,E2 23692.687} C_VEL
LIN {X 0,Y 491.046,Z 1248.074,A -85,B 0,C 180,E1 23690.252,E2 23690.252} C_VEL
LIN {X 0,Y 489.834,Z 1256.148,A -85,B 0,C 180,E1 23687.707,E2 23687.707} C_VEL
LIN {X 0,Y 489.006,Z 1263.043,A -85,B 0,C 180,E1 23685.172,E2 23685.172} C_VEL
LIN {X 0,Y 488.455,Z 1268.814,A -85,B 0,C 180,E1 23682.652,E2 23682.652} C_VEL
LIN {X 0,Y 488.097,Z 1273.923,A -85,B 0,C 180,E1 23679.908,E2 23679.908} C_VEL
LIN {X 0,Y 487.961,Z 1278.283,A -85,B 0,C 180,E1 23676.707,E2 23676.707} C_VEL
LIN {X 0,Y 487.915,Z 1280.674,A -85,B 0,C 180,E1 23673.878,E2 23673.878} C_VEL
LIN {X 0,Y 487.9,Z 1281.735,A -85,B 0,C 180,E1 23671.409,E2 23671.409} C_VEL
LIN {X 0,Y 487.872,Z 1281.825,A -85,B 0,C 180,E1 23669.061,E2 23669.061} C_VEL
LIN {X 0,Y 487.911,Z 1281.013,A -85,B 0,C 180,E1 23666.71,E2 23666.71} C_VEL
LIN {X 0,Y 487.939,Z 1279.19,A -85,B 0,C 180,E1 23664.237,E2 23664.237} C_VEL
LIN {X 0,Y 488.005,Z 1276.336,A -85,B 0,C 180,E1 23661.745,E2 23661.745} C_VEL
LIN {X 0,Y 488.221,Z 1272.27,A -85,B 0,C 180,E1 23659.14,E2 23659.14} C_VEL
LIN {X 0,Y 488.646,Z 1266.78,A -85,B 0,C 180,E1 23656.39,E2 23656.39} C_VEL
LIN {X 0,Y 489.539,Z 1258.617,A -85,B 0,C 180,E1 23653.14,E2 23653.14} C_VEL
LIN {X 0,Y 490.64,Z 1250.502,A -85,B 0,C 180,E1 23650.475,E2 23650.475} C_VEL
LIN {X 0,Y 492.079,Z 1241.965,A -85,B 0,C 180,E1 23648.045,E2 23648.045} C_VEL
LIN {X 0,Y 493.362,Z 1234.224,A -85,B 0,C 180,E1 23646.215,E2 23646.215} C_VEL
LIN {X 0,Y 495.432,Z 1222.379,A -85,B 0,C 180,E1 23643.77,E2 23643.77} C_VEL
LIN {X 0,Y 497.724,Z 1210.472,A -85,B 0,C 180,E1 23641.568,E2 23641.568} C_VEL
LIN {X 0,Y 500.538,Z 1196.484,A -85,B 0,C 180,E1 23639.244,E2 23639.244} C_VEL
LIN {X 0,Y 504.432,Z 1178.346,A -85,B 0,C 180,E1 23636.561,E2 23636.561} C_VEL
LIN {X 0,Y 508.429,Z 1159.989,A -85,B 0,C 180,E1 23634.196,E2 23634.196} C_VEL
LIN {X 0,Y 512.043,Z 1143.828,A -85,B 0,C 180,E1 23632.324,E2 23632.324} C_VEL
LIN {X 0,Y 515.893,Z 1126.639,A -85,B 0,C 180,E1 23630.527,E2 23630.527} C_VEL
LIN {X 0,Y 520.588,Z 1105.715,A -85,B 0,C 180,E1 23628.573,E2 23628.573} C_VEL
LIN {X 0,Y 525.73,Z 1081.797,A -85,B 0,C 180,E1 23626.64,E2 23626.64} C_VEL
LIN {X 0,Y 529.791,Z 1062.273,A -85,B 0,C 180,E1 23625.254,E2 23625.254} C_VEL
LIN {X 0,Y 533.892,Z 1041.669,A -85,B 0,C 180,E1 23623.959,E2 23623.959} C_VEL
LIN {X 0,Y 538.567,Z 1016.844,A -85,B 0,C 180,E1 23622.598,E2 23622.598} C_VEL
LIN {X 0,Y 542.967,Z 990.629,A -85,B 0,C 180,E1 23621.406,E2 23621.406} C_VEL
LIN {X 0,Y 546.275,Z 968.904,A -85,B 0,C 180,E1 23620.571,E2 23620.571} C_VEL
LIN {X 0,Y 549.291,Z 946.758,A -85,B 0,C 180,E1 23619.864,E2 23619.864} C_VEL
LIN {X 0,Y 552.453,Z 919.857,A -85,B 0,C 180,E1 23619.171,E2 23619.171} C_VEL
LIN {X 0,Y 554.699,Z 892.3,A -85,B 0,C 180,E1 23618.644,E2 23618.644} C_VEL
LIN {X 0,Y 565.193,Z 667.856,A -85,B 0,C 180,E1 23615.164,E2 23615.164} C_VEL
LIN {X 0,Y 574.249,Z 495.946,A -85,B 0,C 180,E1 23612.432,E2 23612.432} C_VEL
LIN {X 0,Y 572.453,Z 484.365,A -85,B 0,C 180,E1 23611.896,E2 23611.896} C_VEL
LIN {X 0,Y 561.212,Z 466.841,A -85,B 0,C 180,E1 23609.778,E2 23609.778} C_VEL
LIN {X 0,Y 548.938,Z 448.477,A -85,B 0,C 180,E1 23607.265,E2 23607.265} C_VEL
LIN {X 0,Y 535.032,Z 428.756,A -85,B 0,C 180,E1 23604.13,E2 23604.13} C_VEL
LIN {X 0,Y 523.545,Z 413.09,A -85,B 0,C 180,E1 23601.247,E2 23601.247} C_VEL
LIN {X 0,Y 515.378,Z 402.277,A -85,B 0,C 180,E1 23599.023,E2 23599.023} C_VEL
LIN {X 0,Y 511.698,Z 397.03,A -85,B 0,C 180,E1 23597.866,E2 23597.866} C_VEL
LIN {X 0,Y 508.322,Z 391.462,A -85,B 0,C 180,E1 23596.337,E2 23596.337} C_VEL
LIN {X 0,Y 505.442,Z 386.461,A -85,B 0,C 180,E1 23594.902,E2 23594.902} C_VEL
LIN {X 0,Y 502.407,Z 381.361,A -85,B 0,C 180,E1 23593.348,E2 23593.348} C_VEL
LIN {X 0,Y 500.149,Z 377.378,A -85,B 0,C 180,E1 23592.117,E2 23592.117} C_VEL
LIN {X 0,Y 497.066,Z 372.48,A -85,B 0,C 180,E1 23590.431,E2 23590.431} C_VEL
LIN {X 0,Y 496.345,Z 371.076,A -85,B 0,C 180,E1 23589.977,E2 23589.977} C_VEL
LIN {X 0,Y 493.906,Z 367.481,A -85,B 0,C 180,E1 23588.616,E2 23588.616} C_VEL
LIN {X 0,Y 492.893,Z 365.488,A -85,B 0,C 180,E1 23587.929,E2 23587.929} C_VEL
LIN {X 0,Y 490.53,Z 362.237,A -85,B 0,C 180,E1 23586.555,E2 23586.555} C_VEL
LIN {X 0,Y 489.99,Z 360.381,A -85,B 0,C 180,E1 23585.856,E2 23585.856} C_VEL
LIN {X 0,Y 489.986,Z 360.177,A -85,B 0,C 180,E1 23582.456,E2 23582.456} C_VEL
LIN {X 0,Y 489.994,Z 360.191,A -85,B 0,C 180,E1 23578.831,E2 23578.831} C_VEL
LIN {X 0,Y 489.962,Z 360.194,A -85,B 0,C 180,E1 23575.318,E2 23575.318} C_VEL
LIN {X 0,Y 489.962,Z 360.195,A -85,B 0,C 180,E1 23571.669,E2 23571.669} C_VEL
LIN {X 0,Y 489.991,Z 360.196,A -85,B 0,C 180,E1 23568.106,E2 23568.106} C_VEL
LIN {X 0,Y 489.976,Z 360.197,A -85,B 0,C 180,E1 23564.616,E2 23564.616} C_VEL
LIN {X 0,Y 489.954,Z 360.2,A -85,B 0,C 180,E1 23561.065,E2 23561.065} C_VEL
LIN {X 0,Y 489.978,Z 360.19,A -85,B 0,C 180,E1 23557.567,E2 23557.567} C_VEL
LIN {X 0,Y 489.99,Z 360.184,A -85,B 0,C 180,E1 23553.977,E2 23553.977} C_VEL
LIN {X 0,Y 489.951,Z 360.185,A -85,B 0,C 180,E1 23550.539,E2 23550.539} C_VEL
LIN {X 0,Y 489.955,Z 360.187,A -85,B 0,C 180,E1 23546.983,E2 23546.983} C_VEL
LIN {X 0,Y 489.992,Z 360.184,A -85,B 0,C 180,E1 23543.513,E2 23543.513} C_VEL
LIN {X 0,Y 489.948,Z 360.194,A -85,B 0,C 180,E1 23540.115,E2 23540.115} C_VEL
LIN {X 0,Y 489.946,Z 360.202,A -85,B 0,C 180,E1 23536.547,E2 23536.547} C_VEL
LIN {X 0,Y 489.987,Z 360.198,A -85,B 0,C 180,E1 23533.067,E2 23533.067} C_VEL
LIN {X 0,Y 489.95,Z 360.2,A -85,B 0,C 180,E1 23529.699,E2 23529.699} C_VEL
LIN {X 0,Y 489.935,Z 360.193,A -85,B 0,C 180,E1 23526.143,E2 23526.143} C_VEL
LIN {X 0,Y 489.979,Z 360.184,A -85,B 0,C 180,E1 23522.736,E2 23522.736} C_VEL
LIN {X 0,Y 489.944,Z 360.184,A -85,B 0,C 180,E1 23519.374,E2 23519.374} C_VEL
LIN {X 0,Y 489.931,Z 360.188,A -85,B 0,C 180,E1 23515.837,E2 23515.837} C_VEL
LIN {X 0,Y 489.981,Z 360.189,A -85,B 0,C 180,E1 23512.417,E2 23512.417} C_VEL
LIN {X 0,Y 489.948,Z 360.199,A -85,B 0,C 180,E1 23508.934,E2 23508.934} C_VEL
LIN {X 0,Y 489.923,Z 360.193,A -85,B 0,C 180,E1 23505.507,E2 23505.507} C_VEL
LIN {X 0,Y 489.972,Z 360.186,A -85,B 0,C 180,E1 23502.134,E2 23502.134} C_VEL
LIN {X 0,Y 489.951,Z 360.381,A -85,B 0,C 180,E1 23500.941,E2 23500.941} C_VEL
LIN {X 0,Y 490.249,Z 361.575,A -85,B 0,C 180,E1 23500.558,E2 23500.558} C_VEL
LIN {X 0,Y 492.145,Z 364.775,A -85,B 0,C 180,E1 23499.81,E2 23499.81} C_VEL
LIN {X 0,Y 495.631,Z 367.365,A -85,B 0,C 180,E1 23498.684,E2 23498.684} C_VEL
LIN {X 0,Y 497.718,Z 370.941,A -85,B 0,C 180,E1 23497.938,E2 23497.938} C_VEL
LIN {X 0,Y 501.074,Z 373.704,A -85,B 0,C 180,E1 23496.905,E2 23496.905} C_VEL
LIN {X 0,Y 503.569,Z 377.526,A -85,B 0,C 180,E1 23496.098,E2 23496.098} C_VEL
LIN {X 0,Y 506.559,Z 380.161,A -85,B 0,C 180,E1 23495.238,E2 23495.238} C_VEL
LIN {X 0,Y 509.6,Z 384.334,A -85,B 0,C 180,E1 23494.332,E2 23494.332} C_VEL
LIN {X 0,Y 511.846,Z 386.415,A -85,B 0,C 180,E1 23493.724,E2 23493.724} C_VEL
LIN {X 0,Y 515.39,Z 390.882,A -85,B 0,C 180,E1 23492.746,E2 23492.746} C_VEL
LIN {X 0,Y 517.19,Z 392.941,A -85,B 0,C 180,E1 23492.266,E2 23492.266} C_VEL
LIN {X 0,Y 521.074,Z 397.456,A -85,B 0,C 180,E1 23491.27,E2 23491.27} C_VEL
LIN {X 0,Y 525.946,Z 403.327,A -85,B 0,C 180,E1 23490.077,E2 23490.077} C_VEL
LIN {X 0,Y 532.631,Z 411.624,A -85,B 0,C 180,E1 23488.494,E2 23488.494} C_VEL
LIN {X 0,Y 544.394,Z 426.227,A -85,B 0,C 180,E1 23485.95,E2 23485.95} C_VEL
LIN {X 0,Y 559.636,Z 446.123,A -85,B 0,C 180,E1 23482.97,E2 23482.97} C_VEL
LIN {X 0,Y 571.158,Z 462.225,A -85,B 0,C 180,E1 23480.898,E2 23480.898} C_VEL
LIN {X 0,Y 568.713,Z 507.23,A -85,B 0,C 180,E1 23480.188,E2 23480.188} C_VEL
LIN {X 0,Y 567.705,Z 514.921,A -85,B 0,C 180,E1 23480.148,E2 23480.148} C_VEL
LIN {X 0,Y 562.883,Z 535.533,A -85,B 0,C 180,E1 23480.337,E2 23480.337} C_VEL
LIN {X 0,Y 562.08,Z 542.132,A -85,B 0,C 180,E1 23480.294,E2 23480.294} C_VEL
LIN {X 0,Y 552.125,Z 740.186,A -85,B 0,C 180,E1 23477.211,E2 23477.211} C_VEL
LIN {X 0,Y 549.882,Z 778.597,A -85,B 0,C 180,E1 23476.567,E2 23476.567} C_VEL
LIN {X 0,Y 547.697,Z 802.78,A -85,B 0,C 180,E1 23476.005,E2 23476.005} C_VEL
LIN {X 0,Y 545.231,Z 824.765,A -85,B 0,C 180,E1 23475.363,E2 23475.363} C_VEL
LIN {X 0,Y 542.142,Z 847.887,A -85,B 0,C 180,E1 23474.544,E2 23474.544} C_VEL
LIN {X 0,Y 537.821,Z 875.063,A -85,B 0,C 180,E1 23473.363,E2 23473.363} C_VEL
LIN {X 0,Y 534.027,Z 895.784,A -85,B 0,C 180,E1 23472.292,E2 23472.292} C_VEL
LIN {X 0,Y 530.099,Z 915.355,A -85,B 0,C 180,E1 23471.126,E2 23471.126} C_VEL
LIN {X 0,Y 525.679,Z 935.658,A -85,B 0,C 180,E1 23469.746,E2 23469.746} C_VEL
LIN {X 0,Y 519.979,Z 959.565,A -85,B 0,C 180,E1 23467.859,E2 23467.859} C_VEL
LIN {X 0,Y 515.371,Z 977.738,A -85,B 0,C 180,E1 23466.2,E2 23466.2} C_VEL
LIN {X 0,Y 511.032,Z 994.222,A -85,B 0,C 180,E1 23464.504,E2 23464.504} C_VEL
LIN {X 0,Y 506.287,Z 1011.719,A -85,B 0,C 180,E1 23462.469,E2 23462.469} C_VEL
LIN {X 0,Y 501.039,Z 1030.485,A -85,B 0,C 180,E1 23459.941,E2 23459.941} C_VEL
LIN {X 0,Y 497.243,Z 1044.112,A -85,B 0,C 180,E1 23457.842,E2 23457.842} C_VEL
LIN {X 0,Y 493.672,Z 1057.082,A -85,B 0,C 180,E1 23455.592,E2 23455.592} C_VEL
LIN {X 0,Y 489.972,Z 1070.995,A -85,B 0,C 180,E1 23452.84,E2 23452.84} C_VEL
LIN {X 0,Y 486.725,Z 1083.852,A -85,B 0,C 180,E1 23449.831,E2 23449.831} C_VEL
LIN {X 0,Y 484.209,Z 1094.849,A -85,B 0,C 180,E1 23446.798,E2 23446.798} C_VEL
LIN {X 0,Y 482.326,Z 1104.357,A -85,B 0,C 180,E1 23443.656,E2 23443.656} C_VEL
LIN {X 0,Y 480.948,Z 1114.459,A -85,B 0,C 180,E1 23439.817,E2 23439.817} C_VEL
LIN {X 0,Y 480.352,Z 1120.815,A -85,B 0,C 180,E1 23436.834,E2 23436.834} C_VEL
LIN {X 0,Y 480.048,Z 1125.769,A -85,B 0,C 180,E1 23433.789,E2 23433.789} C_VEL
LIN {X 0,Y 479.941,Z 1129.393,A -85,B 0,C 180,E1 23430.692,E2 23430.692} C_VEL
LIN {X 0,Y 479.903,Z 1131.283,A -85,B 0,C 180,E1 23427.821,E2 23427.821} C_VEL
LIN {X 0,Y 479.894,Z 1131.974,A -85,B 0,C 180,E1 23424.759,E2 23424.759} C_VEL
LIN {X 0,Y 479.924,Z 1131.142,A -85,B 0,C 180,E1 23421.768,E2 23421.768} C_VEL
LIN {X 0,Y 479.946,Z 1128.87,A -85,B 0,C 180,E1 23418.714,E2 23418.714} C_VEL
LIN {X 0,Y 480.072,Z 1125.339,A -85,B 0,C 180,E1 23415.796,E2 23415.796} C_VEL
LIN {X 0,Y 480.418,Z 1119.913,A -85,B 0,C 180,E1 23412.623,E2 23412.623} C_VEL
LIN {X 0,Y 481.087,Z 1113.235,A -85,B 0,C 180,E1 23409.571,E2 23409.571} C_VEL
LIN {X 0,Y 483.205,Z 1100.35,A -85,B 0,C 180,E1 23404.748,E2 23404.748} C_VEL
LIN {X 0,Y 485.617,Z 1090.105,A -85,B 0,C 180,E1 23401.534,E2 23401.534} C_VEL
LIN {X 0,Y 488.528,Z 1078.855,A -85,B 0,C 180,E1 23398.593,E2 23398.593} C_VEL
LIN {X 0,Y 491.368,Z 1068.603,A -85,B 0,C 180,E1 23396.266,E2 23396.266} C_VEL
LIN {X 0,Y 494.72,Z 1057.084,A -85,B 0,C 180,E1 23393.967,E2 23393.967} C_VEL
LIN {X 0,Y 499.367,Z 1041.382,A -85,B 0,C 180,E1 23391.247,E2 23391.247} C_VEL
LIN {X 0,Y 503.73,Z 1026.375,A -85,B 0,C 180,E1 23389.015,E2 23389.015} C_VEL
LIN {X 0,Y 507.823,Z 1012.168,A -85,B 0,C 180,E1 23387.144,E2 23387.144} C_VEL
LIN {X 0,Y 512.819,Z 994.449,A -85,B 0,C 180,E1 23385.086,E2 23385.086} C_VEL
LIN {X 0,Y 518,Z 974.571,A -85,B 0,C 180,E1 23383.112,E2 23383.112} C_VEL
LIN {X 0,Y 521.973,Z 958.313,A -85,B 0,C 180,E1 23381.69,E2 23381.69} C_VEL
LIN {X 0,Y 526.121,Z 940.155,A -85,B 0,C 180,E1 23380.285,E2 23380.285} C_VEL
LIN {X 0,Y 531.062,Z 916.173,A -85,B 0,C 180,E1 23378.692,E2 23378.692} C_VEL
LIN {X 0,Y 534.77,Z 895.403,A -85,B 0,C 180,E1 23377.52,E2 23377.52} C_VEL
LIN {X 0,Y 537.894,Z 875.676,A -85,B 0,C 180,E1 23376.559,E2 23376.559} C_VEL
LIN {X 0,Y 541.294,Z 850.488,A -85,B 0,C 180,E1 23375.521,E2 23375.521} C_VEL
LIN {X 0,Y 543.755,Z 827.504,A -85,B 0,C 180,E1 23374.754,E2 23374.754} C_VEL
LIN {X 0,Y 545.79,Z 803.876,A -85,B 0,C 180,E1 23374.113,E2 23374.113} C_VEL
LIN {X 0,Y 547.923,Z 769.913,A -85,B 0,C 180,E1 23373.432,E2 23373.432} C_VEL
LIN {X 0,Y 553.359,Z 697.428,A -85,B 0,C 180,E1 23372.139,E2 23372.139} C_VEL
LIN {X 0,Y 560.145,Z 630.527,A -85,B 0,C 180,E1 23370.861,E2 23370.861} C_VEL
LIN {X 0,Y 568.009,Z 572.227,A -85,B 0,C 180,E1 23369.691,E2 23369.691} C_VEL
LIN {X 0,Y 577.554,Z 515.42,A -85,B 0,C 180,E1 23368.539,E2 23368.539} C_VEL
LIN {X 0,Y 579.061,Z 507.442,A -85,B 0,C 180,E1 23368.374,E2 23368.374} C_VEL
LIN {X 0,Y 569.12,Z 565.292,A -85,B 0,C 180,E1 23367.17,E2 23367.17} C_VEL
LIN {X 0,Y 560.631,Z 627.587,A -85,B 0,C 180,E1 23365.886,E2 23365.886} C_VEL
LIN {X 0,Y 553.593,Z 696.215,A -85,B 0,C 180,E1 23364.54,E2 23364.54} C_VEL
LIN {X 0,Y 548.025,Z 770.329,A -85,B 0,C 180,E1 23363.183,E2 23363.183} C_VEL
LIN {X 0,Y 541.887,Z 878.355,A -85,B 0,C 180,E1 23361.333,E2 23361.333} C_VEL
LIN {X 0,Y 539.347,Z 906.63,A -85,B 0,C 180,E1 23360.724,E2 23360.724} C_VEL
LIN {X 0,Y 536.123,Z 935.216,A -85,B 0,C 180,E1 23359.979,E2 23359.979} C_VEL
LIN {X 0,Y 532.252,Z 964.924,A -85,B 0,C 180,E1 23359.001,E2 23359.001} C_VEL
LIN {X 0,Y 529.001,Z 988.407,A -85,B 0,C 180,E1 23358.07,E2 23358.07} C_VEL
LIN {X 0,Y 525.291,Z 1013.507,A -85,B 0,C 180,E1 23356.918,E2 23356.918} C_VEL
LIN {X 0,Y 520.559,Z 1043.383,A -85,B 0,C 180,E1 23355.291,E2 23355.291} C_VEL
LIN {X 0,Y 516.845,Z 1065.313,A -85,B 0,C 180,E1 23353.902,E2 23353.902} C_VEL
LIN {X 0,Y 513.401,Z 1084.813,A -85,B 0,C 180,E1 23352.516,E2 23352.516} C_VEL
LIN {X 0,Y 510.015,Z 1103.297,A -85,B 0,C 180,E1 23351.053,E2 23351.053} C_VEL
LIN {X 0,Y 506.589,Z 1121.448,A -85,B 0,C 180,E1 23349.46,E2 23349.46} C_VEL
LIN {X 0,Y 502.982,Z 1140.318,A -85,B 0,C 180,E1 23347.61,E2 23347.61} C_VEL
LIN {X 0,Y 498.61,Z 1162.87,A -85,B 0,C 180,E1 23345.096,E2 23345.096} C_VEL
LIN {X 0,Y 495.391,Z 1179.237,A -85,B 0,C 180,E1 23343.022,E2 23343.022} C_VEL
LIN {X 0,Y 492.668,Z 1193.29,A -85,B 0,C 180,E1 23341.031,E2 23341.031} C_VEL
LIN {X 0,Y 490.393,Z 1205.25,A -85,B 0,C 180,E1 23339.163,E2 23339.163} C_VEL
LIN {X 0,Y 488.309,Z 1216.857,A -85,B 0,C 180,E1 23337.169,E2 23337.169} C_VEL
LIN {X 0,Y 486.276,Z 1228.53,A -85,B 0,C 180,E1 23334.93,E2 23334.93} C_VEL
LIN {X 0,Y 484.551,Z 1238.901,A -85,B 0,C 180,E1 23332.698,E2 23332.698} C_VEL
LIN {X 0,Y 483.174,Z 1248.069,A -85,B 0,C 180,E1 23330.471,E2 23330.471} C_VEL
LIN {X 0,Y 482.208,Z 1254.735,A -85,B 0,C 180,E1 23328.497,E2 23328.497} C_VEL
LIN {X 0,Y 481.211,Z 1262.134,A -85,B 0,C 180,E1 23325.795,E2 23325.795} C_VEL
LIN {X 0,Y 480.566,Z 1268.204,A -85,B 0,C 180,E1 23323.157,E2 23323.157} C_VEL
LIN {X 0,Y 480.206,Z 1272.955,A -85,B 0,C 180,E1 23320.639,E2 23320.639} C_VEL
LIN {X 0,Y 479.979,Z 1276.985,A -85,B 0,C 180,E1 23317.903,E2 23317.903} C_VEL
LIN {X 0,Y 479.923,Z 1280.095,A -85,B 0,C 180,E1 23314.9,E2 23314.9} C_VEL
LIN {X 0,Y 479.908,Z 1281.667,A -85,B 0,C 180,E1 23311.791,E2 23311.791} C_VEL
LIN {X 0,Y 479.867,Z 1281.848,A -85,B 0,C 180,E1 23309.164,E2 23309.164} C_VEL
LIN {X 0,Y 479.911,Z 1281.013,A -85,B 0,C 180,E1 23306.656,E2 23306.656} C_VEL
LIN {X 0,Y 479.942,Z 1279.187,A -85,B 0,C 180,E1 23304.141,E2 23304.141} C_VEL
LIN {X 0,Y 480.014,Z 1276.416,A -85,B 0,C 180,E1 23301.67,E2 23301.67} C_VEL
LIN {X 0,Y 480.231,Z 1272.474,A -85,B 0,C 180,E1 23299.078,E2 23299.078} C_VEL
LIN {X 0,Y 480.632,Z 1267.542,A -85,B 0,C 180,E1 23296.526,E2 23296.526} C_VEL
LIN {X 0,Y 481.483,Z 1260.009,A -85,B 0,C 180,E1 23293.347,E2 23293.347} C_VEL
LIN {X 0,Y 482.655,Z 1251.55,A -85,B 0,C 180,E1 23290.493,E2 23290.493} C_VEL
LIN {X 0,Y 484.136,Z 1241.849,A -85,B 0,C 180,E1 23287.921,E2 23287.921} C_VEL
LIN {X 0,Y 485.965,Z 1231.106,A -85,B 0,C 180,E1 23285.428,E2 23285.428} C_VEL
LIN {X 0,Y 488.169,Z 1219.324,A -85,B 0,C 180,E1 23282.998,E2 23282.998} C_VEL
LIN {X 0,Y 491.228,Z 1204.188,A -85,B 0,C 180,E1 23280.221,E2 23280.221} C_VEL
LIN {X 0,Y 494.93,Z 1187.039,A -85,B 0,C 180,E1 23277.494,E2 23277.494} C_VEL
LIN {X 0,Y 498.316,Z 1171.96,A -85,B 0,C 180,E1 23275.355,E2 23275.355} C_VEL
LIN {X 0,Y 501.787,Z 1156.886,A -85,B 0,C 180,E1 23273.422,E2 23273.422} C_VEL
LIN {X 0,Y 505.711,Z 1140.088,A -85,B 0,C 180,E1 23271.479,E2 23271.479} C_VEL
LIN {X 0,Y 510.867,Z 1118.305,A -85,B 0,C 180,E1 23269.24,E2 23269.24} C_VEL
LIN {X 0,Y 515.718,Z 1096.964,A -85,B 0,C 180,E1 23267.343,E2 23267.343} C_VEL
LIN {X 0,Y 519.857,Z 1078.398,A -85,B 0,C 180,E1 23265.872,E2 23265.872} C_VEL
LIN {X 0,Y 523.85,Z 1059.85,A -85,B 0,C 180,E1 23264.558,E2 23264.558} C_VEL
LIN {X 0,Y 528.248,Z 1038.506,A -85,B 0,C 180,E1 23263.22,E2 23263.22} C_VEL
LIN {X 0,Y 533.448,Z 1011.144,A -85,B 0,C 180,E1 23261.755,E2 23261.755} C_VEL
LIN {X 0,Y 537.364,Z 988.377,A -85,B 0,C 180,E1 23260.738,E2 23260.738} C_VEL
LIN {X 0,Y 540.596,Z 967.659,A -85,B 0,C 180,E1 23259.946,E2 23259.946} C_VEL
LIN {X 0,Y 543.661,Z 945.879,A -85,B 0,C 180,E1 23259.248,E2 23259.248} C_VEL
LIN {X 0,Y 546.919,Z 919.154,A -85,B 0,C 180,E1 23258.556,E2 23258.556} C_VEL
LIN {X 0,Y 549.247,Z 891.561,A -85,B 0,C 180,E1 23258.025,E2 23258.025} C_VEL
LIN {X 0,Y 560.309,Z 666.28,A -85,B 0,C 180,E1 23254.496,E2 23254.496} C_VEL
LIN {X 0,Y 569.519,Z 498.07,A -85,B 0,C 180,E1 23251.81,E2 23251.81} C_VEL
LIN {X 0,Y 568.212,Z 489.494,A -85,B 0,C 180,E1 23251.41,E2 23251.41} C_VEL
LIN {X 0,Y 556.599,Z 471.165,A -85,B 0,C 180,E1 23249.162,E2 23249.162} C_VEL
LIN {X 0,Y 544.431,Z 453.225,A -85,B 0,C 180,E1 23246.624,E2 23246.624} C_VEL
LIN {X 0,Y 533.793,Z 437.922,A -85,B 0,C 180,E1 23244.19,E2 23244.19} C_VEL
LIN {X 0,Y 524.031,Z 424.308,A -85,B 0,C 180,E1 23241.755,E2 23241.755} C_VEL
LIN {X 0,Y 513.398,Z 409.96,A -85,B 0,C 180,E1 23238.863,E2 23238.863} C_VEL
LIN {X 0,Y 508.274,Z 403.269,A -85,B 0,C 180,E1 23237.34,E2 23237.34} C_VEL
LIN {X 0,Y 503.804,Z 397.52,A -85,B 0,C 180,E1 23235.955,E2 23235.955} C_VEL
LIN {X 0,Y 500.937,Z 393.014,A -85,B 0,C 180,E1 23234.803,E2 23234.803} C_VEL
LIN {X 0,Y 497.875,Z 387.88,A -85,B 0,C 180,E1 23233.235,E2 23233.235} C_VEL
LIN {X 0,Y 495.454,Z 383.518,A -85,B 0,C 180,E1 23231.879,E2 23231.879} C_VEL
LIN {X 0,Y 492.567,Z 379.014,A -85,B 0,C 180,E1 23230.29,E2 23230.29} C_VEL
LIN {X 0,Y 491.581,Z 377.347,A -85,B 0,C 180,E1 23229.72,E2 23229.72} C_VEL
LIN {X 0,Y 489.261,Z 373.588,A -85,B 0,C 180,E1 23228.343,E2 23228.343} C_VEL
LIN {X 0,Y 488.381,Z 372.016,A -85,B 0,C 180,E1 23227.766,E2 23227.766} C_VEL
LIN {X 0,Y 486.061,Z 368.699,A -85,B 0,C 180,E1 23226.378,E2 23226.378} C_VEL
LIN {X 0,Y 485.154,Z 366.665,A -85,B 0,C 180,E1 23225.677,E2 23225.677} C_VEL
LIN {X 0,Y 482.545,Z 363.173,A -85,B 0,C 180,E1 23224.04,E2 23224.04} C_VEL
LIN {X 0,Y 482.062,Z 361.387,A -85,B 0,C 180,E1 23223.329,E2 23223.329} C_VEL
LIN {X 0,Y 482.025,Z 361.19,A -85,B 0,C 180,E1 23219.762,E2 23219.762} C_VEL
LIN {X 0,Y 482.043,Z 361.188,A -85,B 0,C 180,E1 23216.124,E2 23216.124} C_VEL
LIN {X 0,Y 482.058,Z 361.183,A -85,B 0,C 180,E1 23212.491,E2 23212.491} C_VEL
LIN {X 0,Y 482.031,Z 361.184,A -85,B 0,C 180,E1 23208.877,E2 23208.877} C_VEL
LIN {X 0,Y 482.015,Z 361.184,A -85,B 0,C 180,E1 23205.34,E2 23205.34} C_VEL
LIN {X 0,Y 482.048,Z 361.178,A -85,B 0,C 180,E1 23201.804,E2 23201.804} C_VEL
LIN {X 0,Y 482.056,Z 361.185,A -85,B 0,C 180,E1 23198.205,E2 23198.205} C_VEL
LIN {X 0,Y 482.015,Z 361.188,A -85,B 0,C 180,E1 23194.702,E2 23194.702} C_VEL
LIN {X 0,Y 482.018,Z 361.177,A -85,B 0,C 180,E1 23191.089,E2 23191.089} C_VEL
LIN {X 0,Y 482.055,Z 361.171,A -85,B 0,C 180,E1 23187.586,E2 23187.586} C_VEL
LIN {X 0,Y 482.023,Z 361.173,A -85,B 0,C 180,E1 23184.052,E2 23184.052} C_VEL
LIN {X 0,Y 482.004,Z 361.178,A -85,B 0,C 180,E1 23180.505,E2 23180.505} C_VEL
LIN {X 0,Y 482.04,Z 361.176,A -85,B 0,C 180,E1 23177.072,E2 23177.072} C_VEL
LIN {X 0,Y 482.042,Z 361.184,A -85,B 0,C 180,E1 23173.448,E2 23173.448} C_VEL
LIN {X 0,Y 482.001,Z 361.192,A -85,B 0,C 180,E1 23170.021,E2 23170.021} C_VEL
LIN {X 0,Y 482.017,Z 361.185,A -85,B 0,C 180,E1 23166.537,E2 23166.537} C_VEL
LIN {X 0,Y 482.041,Z 361.175,A -85,B 0,C 180,E1 23163.061,E2 23163.061} C_VEL
LIN {X 0,Y 481.993,Z 361.175,A -85,B 0,C 180,E1 23159.632,E2 23159.632} C_VEL
LIN {X 0,Y 482.001,Z 361.174,A -85,B 0,C 180,E1 23156.072,E2 23156.072} C_VEL
LIN {X 0,Y 482.057,Z 361.173,A -85,B 0,C 180,E1 23152.565,E2 23152.565} C_VEL
LIN {X 0,Y 482.004,Z 361.189,A -85,B 0,C 180,E1 23149.007,E2 23149.007} C_VEL
LIN {X 0,Y 481.985,Z 361.182,A -85,B 0,C 180,E1 23145.522,E2 23145.522} C_VEL
LIN {X 0,Y 482.032,Z 361.518,A -85,B 0,C 180,E1 23143.434,E2 23143.434} C_VEL
LIN {X 0,Y 482.571,Z 363.327,A -85,B 0,C 180,E1 23142.9,E2 23142.9} C_VEL
LIN {X 0,Y 484.727,Z 366.238,A -85,B 0,C 180,E1 23142.025,E2 23142.025} C_VEL
LIN {X 0,Y 487.762,Z 368.364,A -85,B 0,C 180,E1 23140.963,E2 23140.963} C_VEL
LIN {X 0,Y 489.927,Z 372.043,A -85,B 0,C 180,E1 23140.109,E2 23140.109} C_VEL
LIN {X 0,Y 493.334,Z 374.753,A -85,B 0,C 180,E1 23138.978,E2 23138.978} C_VEL
LIN {X 0,Y 495.777,Z 378.577,A -85,B 0,C 180,E1 23138.116,E2 23138.116} C_VEL
LIN {X 0,Y 498.842,Z 381.235,A -85,B 0,C 180,E1 23137.163,E2 23137.163} C_VEL
LIN {X 0,Y 501.722,Z 385.28,A -85,B 0,C 180,E1 23136.235,E2 23136.235} C_VEL
LIN {X 0,Y 504.266,Z 387.603,A -85,B 0,C 180,E1 23135.496,E2 23135.496} C_VEL
LIN {X 0,Y 507.542,Z 391.894,A -85,B 0,C 180,E1 23134.52,E2 23134.52} C_VEL
LIN {X 0,Y 509.653,Z 394.038,A -85,B 0,C 180,E1 23133.937,E2 23133.937} C_VEL
LIN {X 0,Y 513.587,Z 398.68,A -85,B 0,C 180,E1 23132.861,E2 23132.861} C_VEL
LIN {X 0,Y 518.553,Z 404.652,A -85,B 0,C 180,E1 23131.547,E2 23131.547} C_VEL
LIN {X 0,Y 523.583,Z 410.689,A -85,B 0,C 180,E1 23130.301,E2 23130.301} C_VEL
LIN {X 0,Y 532.979,Z 422.451,A -85,B 0,C 180,E1 23128.092,E2 23128.092} C_VEL
LIN {X 0,Y 542.771,Z 434.871,A -85,B 0,C 180,E1 23125.986,E2 23125.986} C_VEL
LIN {X 0,Y 556.427,Z 452.752,A -85,B 0,C 180,E1 23123.292,E2 23123.292} C_VEL
LIN {X 0,Y 566.249,Z 466.609,A -85,B 0,C 180,E1 23121.488,E2 23121.488} C_VEL
LIN {X 0,Y 562.08,Z 542.132,A -85,B 0,C 180,E1 23120.294,E2 23120.294} C_VEL
LIN {X 0,Y 561.065,Z 549.822,A -85,B 0,C 180,E1 23120.255,E2 23120.255} C_VEL
LIN {X 0,Y 556.171,Z 570.419,A -85,B 0,C 180,E1 23120.445,E2 23120.445} C_VEL
LIN {X 0,Y 555.359,Z 577.017,A -85,B 0,C 180,E1 23120.403,E2 23120.403} C_VEL
LIN {X 0,Y 545.249,Z 770.053,A -85,B 0,C 180,E1 23117.363,E2 23117.363} C_VEL
LIN {X 0,Y 542.844,Z 798.75,A -85,B 0,C 180,E1 23116.75,E2 23116.75} C_VEL
LIN {X 0,Y 540.095,Z 823.039,A -85,B 0,C 180,E1 23116.058,E2 23116.058} C_VEL
LIN {X 0,Y 537.314,Z 843.725,A -85,B 0,C 180,E1 23115.34,E2 23115.34} C_VEL
LIN {X 0,Y 534.023,Z 864.96,A -85,B 0,C 180,E1 23114.47,E2 23114.47} C_VEL
LIN {X 0,Y 529.498,Z 890.659,A -85,B 0,C 180,E1 23113.218,E2 23113.218} C_VEL
LIN {X 0,Y 524.902,Z 913.227,A -85,B 0,C 180,E1 23111.907,E2 23111.907} C_VEL
LIN {X 0,Y 520.966,Z 931.046,A -85,B 0,C 180,E1 23110.724,E2 23110.724} C_VEL
LIN {X 0,Y 516.683,Z 948.998,A -85,B 0,C 180,E1 23109.378,E2 23109.378} C_VEL
LIN {X 0,Y 512.168,Z 966.88,A -85,B 0,C 180,E1 23107.866,E2 23107.866} C_VEL
LIN {X 0,Y 506.512,Z 988.344,A -85,B 0,C 180,E1 23105.787,E2 23105.787} C_VEL
LIN {X 0,Y 501.519,Z 1006.137,A -85,B 0,C 180,E1 23103.79,E2 23103.79} C_VEL
LIN {X 0,Y 497.335,Z 1020.78,A -85,B 0,C 180,E1 23101.937,E2 23101.937} C_VEL
LIN {X 0,Y 493.275,Z 1034.737,A -85,B 0,C 180,E1 23099.956,E2 23099.956} C_VEL
LIN {X 0,Y 489.444,Z 1048.031,A -85,B 0,C 180,E1 23097.834,E2 23097.834} C_VEL
LIN {X 0,Y 485.063,Z 1063.429,A -85,B 0,C 180,E1 23095.037,E2 23095.037} C_VEL
LIN {X 0,Y 481.529,Z 1076.269,A -85,B 0,C 180,E1 23092.293,E2 23092.293} C_VEL
LIN {X 0,Y 478.741,Z 1087.067,A -85,B 0,C 180,E1 23089.65,E2 23089.65} C_VEL
LIN {X 0,Y 476.129,Z 1098.26,A -85,B 0,C 180,E1 23086.429,E2 23086.429} C_VEL
LIN {X 0,Y 474.304,Z 1107.068,A -85,B 0,C 180,E1 23083.34,E2 23083.34} C_VEL
LIN {X 0,Y 473.072,Z 1114.597,A -85,B 0,C 180,E1 23080.14,E2 23080.14} C_VEL
LIN {X 0,Y 472.252,Z 1122.276,A -85,B 0,C 180,E1 23076.209,E2 23076.209} C_VEL
LIN {X 0,Y 472.004,Z 1126.467,A -85,B 0,C 180,E1 23073.421,E2 23073.421} C_VEL
LIN {X 0,Y 471.936,Z 1129.776,A -85,B 0,C 180,E1 23070.282,E2 23070.282} C_VEL
LIN {X 0,Y 471.882,Z 1131.443,A -85,B 0,C 180,E1 23067.512,E2 23067.512} C_VEL
LIN {X 0,Y 471.888,Z 1131.942,A -85,B 0,C 180,E1 23064.539,E2 23064.539} C_VEL
LIN {X 0,Y 471.923,Z 1131.047,A -85,B 0,C 180,E1 23061.503,E2 23061.503} C_VEL
LIN {X 0,Y 471.956,Z 1128.657,A -85,B 0,C 180,E1 23058.402,E2 23058.402} C_VEL
LIN {X 0,Y 472.113,Z 1124.954,A -85,B 0,C 180,E1 23055.352,E2 23055.352} C_VEL
LIN {X 0,Y 472.475,Z 1119.539,A -85,B 0,C 180,E1 23052.218,E2 23052.218} C_VEL
LIN {X 0,Y 473.56,Z 1111.798,A -85,B 0,C 180,E1 23048.377,E2 23048.377} C_VEL
LIN {X 0,Y 475.316,Z 1103.241,A -85,B 0,C 180,E1 23044.948,E2 23044.948} C_VEL
LIN {X 0,Y 477.433,Z 1094.449,A -85,B 0,C 180,E1 23042.04,E2 23042.04} C_VEL
LIN {X 0,Y 480.45,Z 1083.339,A -85,B 0,C 180,E1 23038.927,E2 23038.927} C_VEL
LIN {X 0,Y 483.896,Z 1071.236,A -85,B 0,C 180,E1 23036.09,E2 23036.09} C_VEL
LIN {X 0,Y 487.17,Z 1060.432,A -85,B 0,C 180,E1 23033.873,E2 23033.873} C_VEL
LIN {X 0,Y 490.876,Z 1048.368,A -85,B 0,C 180,E1 23031.685,E2 23031.685} C_VEL
LIN {X 0,Y 495.94,Z 1031.907,A -85,B 0,C 180,E1 23029.075,E2 23029.075} C_VEL
LIN {X 0,Y 500.588,Z 1016.341,A -85,B 0,C 180,E1 23026.955,E2 23026.955} C_VEL
LIN {X 0,Y 504.831,Z 1001.763,A -85,B 0,C 180,E1 23025.197,E2 23025.197} C_VEL
LIN {X 0,Y 509.675,Z 984.524,A -85,B 0,C 180,E1 23023.356,E2 23023.356} C_VEL
LIN {X 0,Y 515.245,Z 963.051,A -85,B 0,C 180,E1 23021.384,E2 23021.384} C_VEL
LIN {X 0,Y 519.495,Z 945.22,A -85,B 0,C 180,E1 23019.964,E2 23019.964} C_VEL
LIN {X 0,Y 523.415,Z 927.431,A -85,B 0,C 180,E1 23018.718,E2 23018.718} C_VEL
LIN {X 0,Y 527.945,Z 904.677,A -85,B 0,C 180,E1 23017.33,E2 23017.33} C_VEL
LIN {X 0,Y 531.662,Z 882.794,A -85,B 0,C 180,E1 23016.209,E2 23016.209} C_VEL
LIN {X 0,Y 534.705,Z 862.118,A -85,B 0,C 180,E1 23015.295,E2 23015.295} C_VEL
LIN {X 0,Y 537.946,Z 836.016,A -85,B 0,C 180,E1 23014.337,E2 23014.337} C_VEL
LIN {X 0,Y 540.307,Z 811.262,A -85,B 0,C 180,E1 23013.619,E2 23013.619} C_VEL
LIN {X 0,Y 542.267,Z 785.112,A -85,B 0,C 180,E1 23013.025,E2 23013.025} C_VEL
LIN {X 0,Y 547.783,Z 716.194,A -85,B 0,C 180,E1 23011.756,E2 23011.756} C_VEL
LIN {X 0,Y 554.622,Z 653.502,A -85,B 0,C 180,E1 23010.535,E2 23010.535} C_VEL
LIN {X 0,Y 562.822,Z 596.2,A -85,B 0,C 180,E1 23009.37,E2 23009.37} C_VEL
LIN {X 0,Y 571.478,Z 547.132,A -85,B 0,C 180,E1 23008.361,E2 23008.361} C_VEL
LIN {X 0,Y 561.237,Z 606.718,A -85,B 0,C 180,E1 23007.111,E2 23007.111} C_VEL
LIN {X 0,Y 553.05,Z 667.122,A -85,B 0,C 180,E1 23005.862,E2 23005.862} C_VEL
LIN {X 0,Y 546.194,Z 734.61,A -85,B 0,C 180,E1 23004.535,E2 23004.535} C_VEL
LIN {X 0,Y 540.346,Z 813.819,A -85,B 0,C 180,E1 23003.094,E2 23003.094} C_VEL
LIN {X 0,Y 536.5,Z 875.133,A -85,B 0,C 180,E1 23002.004,E2 23002.004} C_VEL
LIN {X 0,Y 533.801,Z 903.553,A -85,B 0,C 180,E1 23001.379,E2 23001.379} C_VEL
LIN {X 0,Y 530.147,Z 934.197,A -85,B 0,C 180,E1 23000.57,E2 23000.57} C_VEL
LIN {X 0,Y 526.217,Z 962.732,A -85,B 0,C 180,E1 22999.612,E2 22999.612} C_VEL
LIN {X 0,Y 522.737,Z 986.67,A -85,B 0,C 180,E1 22998.656,E2 22998.656} C_VEL
LIN {X 0,Y 518.785,Z 1012.25,A -85,B 0,C 180,E1 22997.47,E2 22997.47} C_VEL
LIN {X 0,Y 513.933,Z 1041.659,A -85,B 0,C 180,E1 22995.852,E2 22995.852} C_VEL
LIN {X 0,Y 509.801,Z 1065.251,A -85,B 0,C 180,E1 22994.341,E2 22994.341} C_VEL
LIN {X 0,Y 505.409,Z 1089.352,A -85,B 0,C 180,E1 22992.578,E2 22992.578} C_VEL
LIN {X 0,Y 500.739,Z 1113.527,A -85,B 0,C 180,E1 22990.538,E2 22990.538} C_VEL
LIN {X 0,Y 497.008,Z 1132.442,A -85,B 0,C 180,E1 22988.731,E2 22988.731} C_VEL
LIN {X 0,Y 493.7,Z 1148.916,A -85,B 0,C 180,E1 22986.978,E2 22986.978} C_VEL
LIN {X 0,Y 490.639,Z 1164.141,A -85,B 0,C 180,E1 22985.193,E2 22985.193} C_VEL
LIN {X 0,Y 487.638,Z 1178.974,A -85,B 0,C 180,E1 22983.264,E2 22983.264} C_VEL
LIN {X 0,Y 484.928,Z 1192.624,A -85,B 0,C 180,E1 22981.305,E2 22981.305} C_VEL
LIN {X 0,Y 482.598,Z 1204.536,A -85,B 0,C 180,E1 22979.408,E2 22979.408} C_VEL
LIN {X 0,Y 480.461,Z 1216.058,A -85,B 0,C 180,E1 22977.382,E2 22977.382} C_VEL
LIN {X 0,Y 478.605,Z 1226.505,A -85,B 0,C 180,E1 22975.358,E2 22975.358} C_VEL
LIN {X 0,Y 476.82,Z 1236.983,A -85,B 0,C 180,E1 22973.087,E2 22973.087} C_VEL
LIN {X 0,Y 475.314,Z 1246.727,A -85,B 0,C 180,E1 22970.696,E2 22970.696} C_VEL
LIN {X 0,Y 474.109,Z 1255.211,A -85,B 0,C 180,E1 22968.315,E2 22968.315} C_VEL
LIN {X 0,Y 473.367,Z 1261.376,A -85,B 0,C 180,E1 22966.316,E2 22966.316} C_VEL
LIN {X 0,Y 472.701,Z 1267.289,A -85,B 0,C 180,E1 22963.829,E2 22963.829} C_VEL
LIN {X 0,Y 472.265,Z 1272.265,A -85,B 0,C 180,E1 22961.232,E2 22961.232} C_VEL
LIN {X 0,Y 472.049,Z 1276.184,A -85,B 0,C 180,E1 22958.649,E2 22958.649} C_VEL
LIN {X 0,Y 471.949,Z 1279.072,A -85,B 0,C 180,E1 22956.081,E2 22956.081} C_VEL
LIN {X 0,Y 471.913,Z 1280.877,A -85,B 0,C 180,E1 22953.644,E2 22953.644} C_VEL
LIN {X 0,Y 471.888,Z 1281.78,A -85,B 0,C 180,E1 22951.214,E2 22951.214} C_VEL
LIN {X 0,Y 471.881,Z 1281.802,A -85,B 0,C 180,E1 22948.907,E2 22948.907} C_VEL
LIN {X 0,Y 471.912,Z 1280.945,A -85,B 0,C 180,E1 22946.477,E2 22946.477} C_VEL
LIN {X 0,Y 471.946,Z 1279.184,A -85,B 0,C 180,E1 22944.041,E2 22944.041} C_VEL
LIN {X 0,Y 472.039,Z 1276.342,A -85,B 0,C 180,E1 22941.473,E2 22941.473} C_VEL
LIN {X 0,Y 472.252,Z 1272.471,A -85,B 0,C 180,E1 22938.891,E2 22938.891} C_VEL
LIN {X 0,Y 472.681,Z 1267.542,A -85,B 0,C 180,E1 22936.295,E2 22936.295} C_VEL
LIN {X 0,Y 473.295,Z 1262.031,A -85,B 0,C 180,E1 22933.934,E2 22933.934} C_VEL
LIN {X 0,Y 474.166,Z 1254.955,A -85,B 0,C 180,E1 22931.56,E2 22931.56} C_VEL
LIN {X 0,Y 475.737,Z 1244.512,A -85,B 0,C 180,E1 22928.549,E2 22928.549} C_VEL
LIN {X 0,Y 477.951,Z 1231.528,A -85,B 0,C 180,E1 22925.398,E2 22925.398} C_VEL
LIN {X 0,Y 480.244,Z 1219.636,A -85,B 0,C 180,E1 22922.873,E2 22922.873} C_VEL
LIN {X 0,Y 482.7,Z 1207.669,A -85,B 0,C 180,E1 22920.598,E2 22920.598} C_VEL
LIN {X 0,Y 485.636,Z 1194.402,A -85,B 0,C 180,E1 22918.33,E2 22918.33} C_VEL
LIN {X 0,Y 489.7,Z 1177.189,A -85,B 0,C 180,E1 22915.699,E2 22915.699} C_VEL
LIN {X 0,Y 494.293,Z 1157.708,A -85,B 0,C 180,E1 22913.113,E2 22913.113} C_VEL
LIN {X 0,Y 498.152,Z 1141.807,A -85,B 0,C 180,E1 22911.227,E2 22911.227} C_VEL
LIN {X 0,Y 502.334,Z 1124.579,A -85,B 0,C 180,E1 22909.392,E2 22909.392} C_VEL
LIN {X 0,Y 507.583,Z 1102.958,A -85,B 0,C 180,E1 22907.341,E2 22907.341} C_VEL
LIN {X 0,Y 512.996,Z 1079.698,A -85,B 0,C 180,E1 22905.439,E2 22905.439} C_VEL
LIN {X 0,Y 517.37,Z 1060.21,A -85,B 0,C 180,E1 22904.034,E2 22904.034} C_VEL
LIN {X 0,Y 521.611,Z 1040.225,A -85,B 0,C 180,E1 22902.763,E2 22902.763} C_VEL
LIN {X 0,Y 526.321,Z 1016.717,A -85,B 0,C 180,E1 22901.457,E2 22901.457} C_VEL
LIN {X 0,Y 531.172,Z 989.956,A -85,B 0,C 180,E1 22900.216,E2 22900.216} C_VEL
LIN {X 0,Y 534.752,Z 967.951,A -85,B 0,C 180,E1 22899.361,E2 22899.361} C_VEL
LIN {X 0,Y 537.855,Z 946.799,A -85,B 0,C 180,E1 22898.673,E2 22898.673} C_VEL
LIN {X 0,Y 540.713,Z 924.346,A -85,B 0,C 180,E1 22898.073,E2 22898.073} C_VEL
LIN {X 0,Y 543.575,Z 895.433,A -85,B 0,C 180,E1 22897.471,E2 22897.471} C_VEL
LIN {X 0,Y 546.408,Z 841.27,A -85,B 0,C 180,E1 22896.603,E2 22896.603} C_VEL
LIN {X 0,Y 557.201,Z 631.816,A -85,B 0,C 180,E1 22893.301,E2 22893.301} C_VEL
LIN {X 0,Y 564.748,Z 499.754,A -85,B 0,C 180,E1 22891.16,E2 22891.16} C_VEL
LIN {X 0,Y 563.961,Z 494.543,A -85,B 0,C 180,E1 22890.912,E2 22890.912} C_VEL
LIN {X 0,Y 553.016,Z 477.169,A -85,B 0,C 180,E1 22888.747,E2 22888.747} C_VEL
LIN {X 0,Y 540.856,Z 459.101,A -85,B 0,C 180,E1 22886.163,E2 22886.163} C_VEL
LIN {X 0,Y 529.496,Z 442.63,A -85,B 0,C 180,E1 22883.511,E2 22883.511} C_VEL
LIN {X 0,Y 518.395,Z 427.302,A -85,B 0,C 180,E1 22880.669,E2 22880.669} C_VEL
LIN {X 0,Y 510.25,Z 416.29,A -85,B 0,C 180,E1 22878.361,E2 22878.361} C_VEL
LIN {X 0,Y 505.83,Z 410.422,A -85,B 0,C 180,E1 22877.041,E2 22877.041} C_VEL
LIN {X 0,Y 498.16,Z 400.162,A -85,B 0,C 180,E1 22874.531,E2 22874.531} C_VEL
LIN {X 0,Y 493.498,Z 394.262,A -85,B 0,C 180,E1 22872.937,E2 22872.937} C_VEL
LIN {X 0,Y 490.917,Z 390.087,A -85,B 0,C 180,E1 22871.752,E2 22871.752} C_VEL
LIN {X 0,Y 488.027,Z 385.514,A -85,B 0,C 180,E1 22870.149,E2 22870.149} C_VEL
LIN {X 0,Y 486.812,Z 383.588,A -85,B 0,C 180,E1 22869.458,E2 22869.458} C_VEL
LIN {X 0,Y 484.624,Z 379.692,A -85,B 0,C 180,E1 22868.065,E2 22868.065} C_VEL
LIN {X 0,Y 481.421,Z 374.778,A -85,B 0,C 180,E1 22866.08,E2 22866.08} C_VEL
LIN {X 0,Y 480.628,Z 373.172,A -85,B 0,C 180,E1 22865.491,E2 22865.491} C_VEL
LIN {X 0,Y 478.091,Z 369.599,A -85,B 0,C 180,E1 22863.837,E2 22863.837} C_VEL
LIN {X 0,Y 477.032,Z 367.47,A -85,B 0,C 180,E1 22863.004,E2 22863.004} C_VEL
LIN {X 0,Y 474.594,Z 364.114,A -85,B 0,C 180,E1 22861.328,E2 22861.328} C_VEL
LIN {X 0,Y 474.142,Z 362.332,A -85,B 0,C 180,E1 22860.483,E2 22860.483} C_VEL
LIN {X 0,Y 474.107,Z 362.169,A -85,B 0,C 180,E1 22856.857,E2 22856.857} C_VEL
LIN {X 0,Y 474.083,Z 362.172,A -85,B 0,C 180,E1 22853.339,E2 22853.339} C_VEL
LIN {X 0,Y 474.089,Z 362.172,A -85,B 0,C 180,E1 22849.673,E2 22849.673} C_VEL
LIN {X 0,Y 474.121,Z 362.173,A -85,B 0,C 180,E1 22846.089,E2 22846.089} C_VEL
LIN {X 0,Y 474.107,Z 362.159,A -85,B 0,C 180,E1 22842.412,E2 22842.412} C_VEL
LIN {X 0,Y 474.079,Z 362.171,A -85,B 0,C 180,E1 22838.783,E2 22838.783} C_VEL
LIN {X 0,Y 474.077,Z 362.179,A -85,B 0,C 180,E1 22835.05,E2 22835.05} C_VEL
LIN {X 0,Y 474.113,Z 362.169,A -85,B 0,C 180,E1 22831.534,E2 22831.534} C_VEL
LIN {X 0,Y 474.103,Z 362.165,A -85,B 0,C 180,E1 22827.974,E2 22827.974} C_VEL
LIN {X 0,Y 474.069,Z 362.164,A -85,B 0,C 180,E1 22824.399,E2 22824.399} C_VEL
LIN {X 0,Y 474.07,Z 362.165,A -85,B 0,C 180,E1 22820.719,E2 22820.719} C_VEL
LIN {X 0,Y 474.114,Z 362.16,A -85,B 0,C 180,E1 22817.392,E2 22817.392} C_VEL
LIN {X 0,Y 474.078,Z 362.171,A -85,B 0,C 180,E1 22813.771,E2 22813.771} C_VEL
LIN {X 0,Y 474.062,Z 362.181,A -85,B 0,C 180,E1 22810.196,E2 22810.196} C_VEL
LIN {X 0,Y 474.094,Z 362.175,A -85,B 0,C 180,E1 22806.732,E2 22806.732} C_VEL
LIN {X 0,Y 474.099,Z 362.165,A -85,B 0,C 180,E1 22803.109,E2 22803.109} C_VEL
LIN {X 0,Y 474.054,Z 362.164,A -85,B 0,C 180,E1 22799.656,E2 22799.656} C_VEL
LIN {X 0,Y 474.059,Z 362.163,A -85,B 0,C 180,E1 22796.022,E2 22796.022} C_VEL
LIN {X 0,Y 474.104,Z 362.165,A -85,B 0,C 180,E1 22792.441,E2 22792.441} C_VEL
LIN {X 0,Y 474.069,Z 362.176,A -85,B 0,C 180,E1 22788.954,E2 22788.954} C_VEL
LIN {X 0,Y 474.132,Z 362.402,A -85,B 0,C 180,E1 22786.289,E2 22786.289} C_VEL
LIN {X 0,Y 474.45,Z 363.846,A -85,B 0,C 180,E1 22785.775,E2 22785.775} C_VEL
LIN {X 0,Y 476.241,Z 366.734,A -85,B 0,C 180,E1 22784.903,E2 22784.903} C_VEL
LIN {X 0,Y 479.903,Z 369.454,A -85,B 0,C 180,E1 22783.464,E2 22783.464} C_VEL
LIN {X 0,Y 481.901,Z 372.86,A -85,B 0,C 180,E1 22782.583,E2 22782.583} C_VEL
LIN {X 0,Y 485.115,Z 375.346,A -85,B 0,C 180,E1 22781.412,E2 22781.412} C_VEL
LIN {X 0,Y 485.994,Z 376.682,A -85,B 0,C 180,E1 22781.07,E2 22781.07} C_VEL
LIN {X 0,Y 488.652,Z 380.298,A -85,B 0,C 180,E1 22780.076,E2 22780.076} C_VEL
LIN {X 0,Y 491.186,Z 382.351,A -85,B 0,C 180,E1 22779.226,E2 22779.226} C_VEL
LIN {X 0,Y 493.933,Z 386.304,A -85,B 0,C 180,E1 22778.264,E2 22778.264} C_VEL
LIN {X 0,Y 496.672,Z 388.804,A -85,B 0,C 180,E1 22777.403,E2 22777.403} C_VEL
LIN {X 0,Y 499.882,Z 393.017,A -85,B 0,C 180,E1 22776.374,E2 22776.374} C_VEL
LIN {X 0,Y 502.026,Z 395.074,A -85,B 0,C 180,E1 22775.744,E2 22775.744} C_VEL
LIN {X 0,Y 505.624,Z 399.586,A -85,B 0,C 180,E1 22774.667,E2 22774.667} C_VEL
LIN {X 0,Y 507.348,Z 401.464,A -85,B 0,C 180,E1 22774.182,E2 22774.182} C_VEL
LIN {X 0,Y 512.54,Z 407.745,A -85,B 0,C 180,E1 22772.756,E2 22772.756} C_VEL
LIN {X 0,Y 517.514,Z 413.872,A -85,B 0,C 180,E1 22771.439,E2 22771.439} C_VEL
LIN {X 0,Y 522.946,Z 420.38,A -85,B 0,C 180,E1 22770.101,E2 22770.101} C_VEL
LIN {X 0,Y 530.045,Z 429.188,A -85,B 0,C 180,E1 22768.433,E2 22768.433} C_VEL
LIN {X 0,Y 542.129,Z 444.577,A -85,B 0,C 180,E1 22765.822,E2 22765.822} C_VEL
LIN {X 0,Y 554.995,Z 461.914,A -85,B 0,C 180,E1 22763.275,E2 22763.275} C_VEL
LIN {X 0,Y 561.39,Z 471.118,A -85,B 0,C 180,E1 22762.086,E2 22762.086} C_VEL
LIN {X 0,Y 555.359,Z 577.017,A -85,B 0,C 180,E1 22760.403,E2 22760.403} C_VEL
LIN {X 0,Y 554.344,Z 584.705,A -85,B 0,C 180,E1 22760.364,E2 22760.364} C_VEL
LIN {X 0,Y 549.442,Z 605.296,A -85,B 0,C 180,E1 22760.559,E2 22760.559} C_VEL
LIN {X 0,Y 548.607,Z 611.892,A -85,B 0,C 180,E1 22760.517,E2 22760.517} C_VEL
LIN {X 0,Y 539.976,Z 771.37,A -85,B 0,C 180,E1 22757.986,E2 22757.986} C_VEL
LIN {X 0,Y 537.46,Z 800.297,A -85,B 0,C 180,E1 22757.36,E2 22757.36} C_VEL
LIN {X 0,Y 534.69,Z 824.03,A -85,B 0,C 180,E1 22756.678,E2 22756.678} C_VEL
LIN {X 0,Y 531.838,Z 844.65,A -85,B 0,C 180,E1 22755.958,E2 22755.958} C_VEL
LIN {X 0,Y 528.475,Z 865.739,A -85,B 0,C 180,E1 22755.089,E2 22755.089} C_VEL
LIN {X 0,Y 524.022,Z 890.538,A -85,B 0,C 180,E1 22753.882,E2 22753.882} C_VEL
LIN {X 0,Y 519.332,Z 912.971,A -85,B 0,C 180,E1 22752.579,E2 22752.579} C_VEL
LIN {X 0,Y 515.019,Z 931.962,A -85,B 0,C 180,E1 22751.317,E2 22751.317} C_VEL
LIN {X 0,Y 510.617,Z 950.009,A -85,B 0,C 180,E1 22749.96,E2 22749.96} C_VEL
LIN {X 0,Y 505.966,Z 967.945,A -85,B 0,C 180,E1 22748.434,E2 22748.434} C_VEL
LIN {X 0,Y 500.017,Z 989.744,A -85,B 0,C 180,E1 22746.301,E2 22746.301} C_VEL
LIN {X 0,Y 494.905,Z 1007.369,A -85,B 0,C 180,E1 22744.302,E2 22744.302} C_VEL
LIN {X 0,Y 490.607,Z 1021.92,A -85,B 0,C 180,E1 22742.443,E2 22742.443} C_VEL
LIN {X 0,Y 486.403,Z 1035.93,A -85,B 0,C 180,E1 22740.439,E2 22740.439} C_VEL
LIN {X 0,Y 482.001,Z 1050.697,A -85,B 0,C 180,E1 22738.044,E2 22738.044} C_VEL
LIN {X 0,Y 477.366,Z 1066.225,A -85,B 0,C 180,E1 22735.123,E2 22735.123} C_VEL
LIN {X 0,Y 474.147,Z 1077.546,A -85,B 0,C 180,E1 22732.658,E2 22732.658} C_VEL
LIN {X 0,Y 471.409,Z 1087.636,A -85,B 0,C 180,E1 22730.16,E2 22730.16} C_VEL
LIN {X 0,Y 468.806,Z 1098.203,A -85,B 0,C 180,E1 22727.128,E2 22727.128} C_VEL
LIN {X 0,Y 466.702,Z 1107.774,A -85,B 0,C 180,E1 22723.79,E2 22723.79} C_VEL
LIN {X 0,Y 465.37,Z 1115.169,A -85,B 0,C 180,E1 22720.673,E2 22720.673} C_VEL
LIN {X 0,Y 464.52,Z 1121.046,A -85,B 0,C 180,E1 22717.529,E2 22717.529} C_VEL
LIN {X 0,Y 464.09,Z 1125.774,A -85,B 0,C 180,E1 22714.175,E2 22714.175} C_VEL
LIN {X 0,Y 463.943,Z 1129.539,A -85,B 0,C 180,E1 22710.693,E2 22710.693} C_VEL
LIN {X 0,Y 463.908,Z 1131.295,A -85,B 0,C 180,E1 22707.886,E2 22707.886} C_VEL
LIN {X 0,Y 463.893,Z 1131.969,A -85,B 0,C 180,E1 22704.718,E2 22704.718} C_VEL
LIN {X 0,Y 463.924,Z 1131.172,A -85,B 0,C 180,E1 22701.734,E2 22701.734} C_VEL
LIN {X 0,Y 463.953,Z 1128.883,A -85,B 0,C 180,E1 22698.513,E2 22698.513} C_VEL
LIN {X 0,Y 464.211,Z 1124.459,A -85,B 0,C 180,E1 22694.597,E2 22694.597} C_VEL
LIN {X 0,Y 464.807,Z 1119.687,A -85,B 0,C 180,E1 22691.415,E2 22691.415} C_VEL
LIN {X 0,Y 465.934,Z 1113.051,A -85,B 0,C 180,E1 22688.018,E2 22688.018} C_VEL
LIN {X 0,Y 467.733,Z 1104.762,A -85,B 0,C 180,E1 22684.66,E2 22684.66} C_VEL
LIN {X 0,Y 469.753,Z 1096.751,A -85,B 0,C 180,E1 22681.952,E2 22681.952} C_VEL
LIN {X 0,Y 472.185,Z 1088,A -85,B 0,C 180,E1 22679.393,E2 22679.393} C_VEL
LIN {X 0,Y 475.956,Z 1075.506,A -85,B 0,C 180,E1 22676.266,E2 22676.266} C_VEL
LIN {X 0,Y 479.805,Z 1063.187,A -85,B 0,C 180,E1 22673.659,E2 22673.659} C_VEL
LIN {X 0,Y 483.625,Z 1051.271,A -85,B 0,C 180,E1 22671.439,E2 22671.439} C_VEL
LIN {X 0,Y 488.127,Z 1037.253,A -85,B 0,C 180,E1 22669.137,E2 22669.137} C_VEL
LIN {X 0,Y 493.634,Z 1019.673,A -85,B 0,C 180,E1 22666.649,E2 22666.649} C_VEL
LIN {X 0,Y 498.281,Z 1004.335,A -85,B 0,C 180,E1 22664.759,E2 22664.759} C_VEL
LIN {X 0,Y 503.121,Z 987.721,A -85,B 0,C 180,E1 22662.954,E2 22662.954} C_VEL
LIN {X 0,Y 509.025,Z 965.929,A -85,B 0,C 180,E1 22660.91,E2 22660.91} C_VEL
LIN {X 0,Y 513.413,Z 948.263,A -85,B 0,C 180,E1 22659.479,E2 22659.479} C_VEL
LIN {X 0,Y 517.636,Z 929.925,A -85,B 0,C 180,E1 22658.171,E2 22658.171} C_VEL
LIN {X 0,Y 522.537,Z 906.118,A -85,B 0,C 180,E1 22656.705,E2 22656.705} C_VEL
LIN {X 0,Y 526.344,Z 884.709,A -85,B 0,C 180,E1 22655.595,E2 22655.595} C_VEL
LIN {X 0,Y 529.697,Z 863.049,A -85,B 0,C 180,E1 22654.627,E2 22654.627} C_VEL
LIN {X 0,Y 533.162,Z 835.949,A -85,B 0,C 180,E1 22653.633,E2 22653.633} C_VEL
LIN {X 0,Y 535.541,Z 812.974,A -85,B 0,C 180,E1 22652.957,E2 22652.957} C_VEL
LIN {X 0,Y 538.008,Z 782.126,A -85,B 0,C 180,E1 22652.254,E2 22652.254} C_VEL
LIN {X 0,Y 544.372,Z 715.59,A -85,B 0,C 180,E1 22650.982,E2 22650.982} C_VEL
LIN {X 0,Y 552.107,Z 655.685,A -85,B 0,C 180,E1 22649.774,E2 22649.774} C_VEL
LIN {X 0,Y 561.247,Z 600.691,A -85,B 0,C 180,E1 22648.638,E2 22648.638} C_VEL
LIN {X 0,Y 563.808,Z 587.202,A -85,B 0,C 180,E1 22648.347,E2 22648.347} C_VEL
LIN {X 0,Y 554.205,Z 642.266,A -85,B 0,C 180,E1 22647.182,E2 22647.182} C_VEL
LIN {X 0,Y 546.468,Z 698.219,A -85,B 0,C 180,E1 22646.017,E2 22646.017} C_VEL
LIN {X 0,Y 540.269,Z 756.674,A -85,B 0,C 180,E1 22644.852,E2 22644.852} C_VEL
LIN {X 0,Y 534.531,Z 828.368,A -85,B 0,C 180,E1 22643.516,E2 22643.516} C_VEL
LIN {X 0,Y 531.079,Z 874.889,A -85,B 0,C 180,E1 22642.642,E2 22642.642} C_VEL
LIN {X 0,Y 527.92,Z 905.034,A -85,B 0,C 180,E1 22641.951,E2 22641.951} C_VEL
LIN {X 0,Y 523.661,Z 937.265,A -85,B 0,C 180,E1 22641.046,E2 22641.046} C_VEL
LIN {X 0,Y 520.081,Z 961.999,A -85,B 0,C 180,E1 22640.192,E2 22640.192} C_VEL
LIN {X 0,Y 516.378,Z 986.197,A -85,B 0,C 180,E1 22639.209,E2 22639.209} C_VEL
LIN {X 0,Y 511.572,Z 1015.75,A -85,B 0,C 180,E1 22637.796,E2 22637.796} C_VEL
LIN {X 0,Y 507.141,Z 1041.211,A -85,B 0,C 180,E1 22636.35,E2 22636.35} C_VEL
LIN {X 0,Y 503.19,Z 1062.975,A -85,B 0,C 180,E1 22634.945,E2 22634.945} C_VEL
LIN {X 0,Y 498.481,Z 1088.007,A -85,B 0,C 180,E1 22633.102,E2 22633.102} C_VEL
LIN {X 0,Y 493.794,Z 1111.459,A -85,B 0,C 180,E1 22631.101,E2 22631.101} C_VEL
LIN {X 0,Y 490.097,Z 1129.637,A -85,B 0,C 180,E1 22629.355,E2 22629.355} C_VEL
LIN {X 0,Y 486.531,Z 1146.929,A -85,B 0,C 180,E1 22627.506,E2 22627.506} C_VEL
LIN {X 0,Y 483.328,Z 1162.253,A -85,B 0,C 180,E1 22625.689,E2 22625.689} C_VEL
LIN {X 0,Y 480.289,Z 1176.934,A -85,B 0,C 180,E1 22623.769,E2 22623.769} C_VEL
LIN {X 0,Y 477.431,Z 1190.79,A -85,B 0,C 180,E1 22621.756,E2 22621.756} C_VEL
LIN {X 0,Y 474.967,Z 1203.078,A -85,B 0,C 180,E1 22619.789,E2 22619.789} C_VEL
LIN {X 0,Y 472.747,Z 1214.654,A -85,B 0,C 180,E1 22617.73,E2 22617.73} C_VEL
LIN {X 0,Y 470.818,Z 1225.081,A -85,B 0,C 180,E1 22615.673,E2 22615.673} C_VEL
LIN {X 0,Y 469.092,Z 1235.06,A -85,B 0,C 180,E1 22613.49,E2 22613.49} C_VEL
LIN {X 0,Y 467.61,Z 1244.433,A -85,B 0,C 180,E1 22611.184,E2 22611.184} C_VEL
LIN {X 0,Y 466.354,Z 1253.069,A -85,B 0,C 180,E1 22608.76,E2 22608.76} C_VEL
LIN {X 0,Y 465.414,Z 1260.517,A -85,B 0,C 180,E1 22606.346,E2 22606.346} C_VEL
LIN {X 0,Y 464.7,Z 1267.133,A -85,B 0,C 180,E1 22603.818,E2 22603.818} C_VEL
LIN {X 0,Y 464.327,Z 1271.743,A -85,B 0,C 180,E1 22601.678,E2 22601.678} C_VEL
LIN {X 0,Y 464.052,Z 1275.702,A -85,B 0,C 180,E1 22599.175,E2 22599.175} C_VEL
LIN {X 0,Y 463.961,Z 1278.842,A -85,B 0,C 180,E1 22596.434,E2 22596.434} C_VEL
LIN {X 0,Y 463.915,Z 1280.809,A -85,B 0,C 180,E1 22593.831,E2 22593.831} C_VEL
LIN {X 0,Y 463.896,Z 1281.757,A -85,B 0,C 180,E1 22591.359,E2 22591.359} C_VEL
LIN {X 0,Y 463.882,Z 1281.802,A -85,B 0,C 180,E1 22588.888,E2 22588.888} C_VEL
LIN {X 0,Y 463.913,Z 1280.944,A -85,B 0,C 180,E1 22586.416,E2 22586.416} C_VEL
LIN {X 0,Y 463.949,Z 1279.181,A -85,B 0,C 180,E1 22583.938,E2 22583.938} C_VEL
LIN {X 0,Y 464.051,Z 1276.339,A -85,B 0,C 180,E1 22581.325,E2 22581.325} C_VEL
LIN {X 0,Y 464.25,Z 1272.844,A -85,B 0,C 180,E1 22578.949,E2 22578.949} C_VEL
LIN {X 0,Y 464.576,Z 1268.632,A -85,B 0,C 180,E1 22576.813,E2 22576.813} C_VEL
LIN {X 0,Y 465.245,Z 1262.164,A -85,B 0,C 180,E1 22574.161,E2 22574.161} C_VEL
LIN {X 0,Y 466.136,Z 1254.848,A -85,B 0,C 180,E1 22571.62,E2 22571.62} C_VEL
LIN {X 0,Y 467.411,Z 1246.363,A -85,B 0,C 180,E1 22569.069,E2 22569.069} C_VEL
LIN {X 0,Y 469.052,Z 1236.641,A -85,B 0,C 180,E1 22566.508,E2 22566.508} C_VEL
LIN {X 0,Y 471.623,Z 1223.316,A -85,B 0,C 180,E1 22563.427,E2 22563.427} C_VEL
LIN {X 0,Y 474.641,Z 1209.062,A -85,B 0,C 180,E1 22560.604,E2 22560.604} C_VEL
LIN {X 0,Y 477.602,Z 1196.043,A -85,B 0,C 180,E1 22558.3,E2 22558.3} C_VEL
LIN {X 0,Y 481.009,Z 1181.832,A -85,B 0,C 180,E1 22556.039,E2 22556.039} C_VEL
LIN {X 0,Y 484.901,Z 1166.179,A -85,B 0,C 180,E1 22553.804,E2 22553.804} C_VEL
LIN {X 0,Y 490.332,Z 1144.566,A -85,B 0,C 180,E1 22551.092,E2 22551.092} C_VEL
LIN {X 0,Y 494.971,Z 1126.127,A -85,B 0,C 180,E1 22549.071,E2 22549.071} C_VEL
LIN {X 0,Y 499.414,Z 1108.419,A -85,B 0,C 180,E1 22547.335,E2 22547.335} C_VEL
LIN {X 0,Y 504.338,Z 1088.406,A -85,B 0,C 180,E1 22545.586,E2 22545.586} C_VEL
LIN {X 0,Y 510.449,Z 1062.445,A -85,B 0,C 180,E1 22543.632,E2 22543.632} C_VEL
LIN {X 0,Y 515,Z 1041.857,A -85,B 0,C 180,E1 22542.293,E2 22542.293} C_VEL
LIN {X 0,Y 519.179,Z 1021.831,A -85,B 0,C 180,E1 22541.147,E2 22541.147} C_VEL
LIN {X 0,Y 523.402,Z 1000.273,A -85,B 0,C 180,E1 22540.076,E2 22540.076} C_VEL
LIN {X 0,Y 528.253,Z 972.827,A -85,B 0,C 180,E1 22538.928,E2 22538.928} C_VEL
LIN {X 0,Y 532.014,Z 948.353,A -85,B 0,C 180,E1 22538.104,E2 22538.104} C_VEL
LIN {X 0,Y 534.929,Z 926.475,A -85,B 0,C 180,E1 22537.504,E2 22537.504} C_VEL
LIN {X 0,Y 537.533,Z 902.686,A -85,B 0,C 180,E1 22536.984,E2 22536.984} C_VEL
LIN {X 0,Y 539.911,Z 865.711,A -85,B 0,C 180,E1 22536.349,E2 22536.349} C_VEL
LIN {X 0,Y 550.419,Z 665.826,A -85,B 0,C 180,E1 22533.186,E2 22533.186} C_VEL
LIN {X 0,Y 560.119,Z 501.911,A -85,B 0,C 180,E1 22530.522,E2 22530.522} C_VEL
LIN {X 0,Y 559.6,Z 499.297,A -85,B 0,C 180,E1 22530.376,E2 22530.376} C_VEL
LIN {X 0,Y 548.066,Z 481.086,A -85,B 0,C 180,E1 22528.05,E2 22528.05} C_VEL
LIN {X 0,Y 535.398,Z 462.038,A -85,B 0,C 180,E1 22525.261,E2 22525.261} C_VEL
LIN {X 0,Y 523.096,Z 444.366,A -85,B 0,C 180,E1 22522.269,E2 22522.269} C_VEL
LIN {X 0,Y 514.264,Z 432.408,A -85,B 0,C 180,E1 22519.952,E2 22519.952} C_VEL
LIN {X 0,Y 508.019,Z 423.672,A -85,B 0,C 180,E1 22518.118,E2 22518.118} C_VEL
LIN {X 0,Y 503.053,Z 417.149,A -85,B 0,C 180,E1 22516.632,E2 22516.632} C_VEL
LIN {X 0,Y 495.832,Z 407.419,A -85,B 0,C 180,E1 22514.242,E2 22514.242} C_VEL
LIN {X 0,Y 491.088,Z 401.337,A -85,B 0,C 180,E1 22512.583,E2 22512.583} C_VEL
LIN {X 0,Y 487.285,Z 396.247,A -85,B 0,C 180,E1 22511.121,E2 22511.121} C_VEL
LIN {X 0,Y 483.713,Z 391.473,A -85,B 0,C 180,E1 22509.729,E2 22509.729} C_VEL
LIN {X 0,Y 480.571,Z 387.305,A -85,B 0,C 180,E1 22508.254,E2 22508.254} C_VEL
LIN {X 0,Y 479.594,Z 385.278,A -85,B 0,C 180,E1 22507.547,E2 22507.547} C_VEL
LIN {X 0,Y 477.054,Z 381.568,A -85,B 0,C 180,E1 22506.016,E2 22506.016} C_VEL
LIN {X 0,Y 476.096,Z 379.665,A -85,B 0,C 180,E1 22505.302,E2 22505.302} C_VEL
LIN {X 0,Y 473.633,Z 376.018,A -85,B 0,C 180,E1 22503.631,E2 22503.631} C_VEL
LIN {X 0,Y 472.718,Z 374.169,A -85,B 0,C 180,E1 22502.91,E2 22502.91} C_VEL
LIN {X 0,Y 470.296,Z 370.826,A -85,B 0,C 180,E1 22501.218,E2 22501.218} C_VEL
LIN {X 0,Y 469.271,Z 368.608,A -85,B 0,C 180,E1 22500.244,E2 22500.244} C_VEL
LIN {X 0,Y 466.702,Z 365.197,A -85,B 0,C 180,E1 22498.281,E2 22498.281} C_VEL
LIN {X 0,Y 466.175,Z 363.377,A -85,B 0,C 180,E1 22497.418,E2 22497.418} C_VEL
LIN {X 0,Y 466.154,Z 363.163,A -85,B 0,C 180,E1 22493.843,E2 22493.843} C_VEL
LIN {X 0,Y 466.177,Z 363.164,A -85,B 0,C 180,E1 22490.244,E2 22490.244} C_VEL
LIN {X 0,Y 466.167,Z 363.162,A -85,B 0,C 180,E1 22486.606,E2 22486.606} C_VEL
LIN {X 0,Y 466.137,Z 363.151,A -85,B 0,C 180,E1 22483.038,E2 22483.038} C_VEL
LIN {X 0,Y 466.146,Z 363.152,A -85,B 0,C 180,E1 22479.403,E2 22479.403} C_VEL
LIN {X 0,Y 466.177,Z 363.149,A -85,B 0,C 180,E1 22475.95,E2 22475.95} C_VEL
LIN {X 0,Y 466.154,Z 363.163,A -85,B 0,C 180,E1 22472.26,E2 22472.26} C_VEL
LIN {X 0,Y 466.134,Z 363.168,A -85,B 0,C 180,E1 22468.727,E2 22468.727} C_VEL
LIN {X 0,Y 466.145,Z 363.158,A -85,B 0,C 180,E1 22465.06,E2 22465.06} C_VEL
LIN {X 0,Y 466.183,Z 363.147,A -85,B 0,C 180,E1 22461.38,E2 22461.38} C_VEL
LIN {X 0,Y 466.145,Z 363.15,A -85,B 0,C 180,E1 22457.825,E2 22457.825} C_VEL
LIN {X 0,Y 466.124,Z 363.156,A -85,B 0,C 180,E1 22454.199,E2 22454.199} C_VEL
LIN {X 0,Y 466.134,Z 363.161,A -85,B 0,C 180,E1 22450.538,E2 22450.538} C_VEL
LIN {X 0,Y 466.172,Z 363.164,A -85,B 0,C 180,E1 22447.064,E2 22447.064} C_VEL
LIN {X 0,Y 466.134,Z 363.162,A -85,B 0,C 180,E1 22443.443,E2 22443.443} C_VEL
LIN {X 0,Y 466.114,Z 363.154,A -85,B 0,C 180,E1 22439.846,E2 22439.846} C_VEL
LIN {X 0,Y 466.144,Z 363.147,A -85,B 0,C 180,E1 22436.36,E2 22436.36} C_VEL
LIN {X 0,Y 466.167,Z 363.149,A -85,B 0,C 180,E1 22432.711,E2 22432.711} C_VEL
LIN {X 0,Y 466.138,Z 363.372,A -85,B 0,C 180,E1 22429.55,E2 22429.55} C_VEL
LIN {X 0,Y 466.462,Z 364.65,A -85,B 0,C 180,E1 22428.95,E2 22428.95} C_VEL
LIN {X 0,Y 468.466,Z 367.887,A -85,B 0,C 180,E1 22427.835,E2 22427.835} C_VEL
LIN {X 0,Y 472.016,Z 370.345,A -85,B 0,C 180,E1 22426.271,E2 22426.271} C_VEL
LIN {X 0,Y 473.974,Z 373.876,A -85,B 0,C 180,E1 22425.289,E2 22425.289} C_VEL
LIN {X 0,Y 477.805,Z 376.904,A -85,B 0,C 180,E1 22423.74,E2 22423.74} C_VEL
LIN {X 0,Y 480.096,Z 380.544,A -85,B 0,C 180,E1 22422.754,E2 22422.754} C_VEL
LIN {X 0,Y 483.522,Z 383.471,A -85,B 0,C 180,E1 22421.478,E2 22421.478} C_VEL
LIN {X 0,Y 486.267,Z 387.45,A -85,B 0,C 180,E1 22420.425,E2 22420.425} C_VEL
LIN {X 0,Y 489.064,Z 389.903,A -85,B 0,C 180,E1 22419.473,E2 22419.473} C_VEL
LIN {X 0,Y 492.201,Z 394.124,A -85,B 0,C 180,E1 22418.377,E2 22418.377} C_VEL
LIN {X 0,Y 494.414,Z 396.192,A -85,B 0,C 180,E1 22417.67,E2 22417.67} C_VEL
LIN {X 0,Y 497.844,Z 400.557,A -85,B 0,C 180,E1 22416.574,E2 22416.574} C_VEL
LIN {X 0,Y 499.847,Z 402.627,A -85,B 0,C 180,E1 22415.971,E2 22415.971} C_VEL
LIN {X 0,Y 503.723,Z 407.282,A -85,B 0,C 180,E1 22414.811,E2 22414.811} C_VEL
LIN {X 0,Y 510.181,Z 415.107,A -85,B 0,C 180,E1 22413.005,E2 22413.005} C_VEL
LIN {X 0,Y 515.102,Z 421.183,A -85,B 0,C 180,E1 22411.694,E2 22411.694} C_VEL
LIN {X 0,Y 520.812,Z 428.086,A -85,B 0,C 180,E1 22410.27,E2 22410.27} C_VEL
LIN {X 0,Y 527.694,Z 436.745,A -85,B 0,C 180,E1 22408.643,E2 22408.643} C_VEL
LIN {X 0,Y 537.128,Z 448.859,A -85,B 0,C 180,E1 22406.558,E2 22406.558} C_VEL
LIN {X 0,Y 550.349,Z 466.512,A -85,B 0,C 180,E1 22403.875,E2 22403.875} C_VEL
LIN {X 0,Y 556.562,Z 475.387,A -85,B 0,C 180,E1 22402.695,E2 22402.695} C_VEL
LIN {X 0,Y 548.607,Z 611.892,A -85,B 0,C 180,E1 22400.517,E2 22400.517} C_VEL
LIN {X 0,Y 547.549,Z 619.577,A -85,B 0,C 180,E1 22400.478,E2 22400.478} C_VEL
LIN {X 0,Y 542.546,Z 640.145,A -85,B 0,C 180,E1 22400.672,E2 22400.672} C_VEL
LIN {X 0,Y 541.721,Z 646.742,A -85,B 0,C 180,E1 22400.63,E2 22400.63} C_VEL
LIN {X 0,Y 534.727,Z 772.341,A -85,B 0,C 180,E1 22398.623,E2 22398.623} C_VEL
LIN {X 0,Y 532.102,Z 801.549,A -85,B 0,C 180,E1 22397.984,E2 22397.984} C_VEL
LIN {X 0,Y 529.294,Z 825.088,A -85,B 0,C 180,E1 22397.304,E2 22397.304} C_VEL
LIN {X 0,Y 526.24,Z 846.629,A -85,B 0,C 180,E1 22396.546,E2 22396.546} C_VEL
LIN {X 0,Y 522.425,Z 869.903,A -85,B 0,C 180,E1 22395.571,E2 22395.571} C_VEL
LIN {X 0,Y 517.38,Z 896.029,A -85,B 0,C 180,E1 22394.247,E2 22394.247} C_VEL
